LIN {X 0,Y 573.544,Z 345.432,A -85,B 0,C 180,E1 -2260.853,E2 -2260.853} C_VEL
LIN {X 0,Y 573.651,Z 334.309,A -85,B 0,C 180,E1 -2261.446,E2 -2261.446} C_VEL
LIN {X 0,Y 573.758,Z 321.17,A -85,B 0,C 180,E1 -2261.974,E2 -2261.974} C_VEL
LIN {X 0,Y 573.833,Z 308.518,A -85,B 0,C 180,E1 -2262.331,E2 -2262.331} C_VEL
LIN {X 0,Y 573.943,Z 295.311,A -85,B 0,C 180,E1 -2262.553,E2 -2262.553} C_VEL
LIN {X 0,Y 573.985,Z 198.721,A -85,B 0,C 180,E1 -2263.768,E2 -2263.768} C_VEL
LIN {X 0,Y 573.396,Z 194.613,A -85,B 0,C 180,E1 -2263.851,E2 -2263.851} C_VEL
LIN {X 0,Y 573.568,Z 174.153,A -85,B 0,C 180,E1 -2266.722,E2 -2266.722} C_VEL
LIN {X 0,Y 573.786,Z 153.399,A -85,B 0,C 180,E1 -2269.647,E2 -2269.647} C_VEL
LIN {X 0,Y 573.952,Z 134.662,A -85,B 0,C 180,E1 -2272.308,E2 -2272.308} C_VEL
LIN {X 0,Y 573.639,Z 129.359,A -85,B 0,C 180,E1 -2273.082,E2 -2273.082} C_VEL
LIN {X 0,Y 573.228,Z 127.085,A -85,B 0,C 180,E1 -2273.438,E2 -2273.438} C_VEL
LIN {X 0,Y 573.239,Z 127.079,A -85,B 0,C 180,E1 -2276.191,E2 -2276.191} C_VEL
LIN {X 0,Y 573.199,Z 127.081,A -85,B 0,C 180,E1 -2278.567,E2 -2278.567} C_VEL
LIN {X 0,Y 573.219,Z 127.08,A -85,B 0,C 180,E1 -2280.994,E2 -2280.994} C_VEL
LIN {X 0,Y 573.244,Z 127.083,A -85,B 0,C 180,E1 -2283.521,E2 -2283.521} C_VEL
LIN {X 0,Y 573.188,Z 127.082,A -85,B 0,C 180,E1 -2286.054,E2 -2286.054} C_VEL
LIN {X 0,Y 573.23,Z 127.078,A -85,B 0,C 180,E1 -2288.703,E2 -2288.703} C_VEL
LIN {X 0,Y 573.198,Z 127.084,A -85,B 0,C 180,E1 -2291.589,E2 -2291.589} C_VEL
LIN {X 0,Y 573.21,Z 127.081,A -85,B 0,C 180,E1 -2294.673,E2 -2294.673} C_VEL
LIN {X 0,Y 573.203,Z 127.081,A -85,B 0,C 180,E1 -2297.596,E2 -2297.596} C_VEL
LIN {X 0,Y 573.224,Z 127.081,A -85,B 0,C 180,E1 -2300.571,E2 -2300.571} C_VEL
LIN {X 0,Y 573.22,Z 127.083,A -85,B 0,C 180,E1 -2303.075,E2 -2303.075} C_VEL
LIN {X 0,Y 573.221,Z 127.076,A -85,B 0,C 180,E1 -2305.668,E2 -2305.668} C_VEL
LIN {X 0,Y 573.208,Z 127.081,A -85,B 0,C 180,E1 -2308.182,E2 -2308.182} C_VEL
LIN {X 0,Y 573.215,Z 127.087,A -85,B 0,C 180,E1 -2310.631,E2 -2310.631} C_VEL
LIN {X 0,Y 573.195,Z 127.079,A -85,B 0,C 180,E1 -2313.517,E2 -2313.517} C_VEL
LIN {X 0,Y 573.192,Z 127.085,A -85,B 0,C 180,E1 -2316.132,E2 -2316.132} C_VEL
LIN {X 0,Y 573.22,Z 127.077,A -85,B 0,C 180,E1 -2319.172,E2 -2319.172} C_VEL
LIN {X 0,Y 573.2,Z 127.087,A -85,B 0,C 180,E1 -2322.15,E2 -2322.15} C_VEL
LIN {X 0,Y 573.217,Z 127.077,A -85,B 0,C 180,E1 -2325.079,E2 -2325.079} C_VEL
LIN {X 0,Y 573.238,Z 127.082,A -85,B 0,C 180,E1 -2327.97,E2 -2327.97} C_VEL
LIN {X 0,Y 573.221,Z 127.076,A -85,B 0,C 180,E1 -2330.828,E2 -2330.828} C_VEL
LIN {X 0,Y 573.233,Z 127.081,A -85,B 0,C 180,E1 -2333.665,E2 -2333.665} C_VEL
LIN {X 0,Y 573.22,Z 127.085,A -85,B 0,C 180,E1 -2335.781,E2 -2335.781} C_VEL
LIN {X 0,Y 573.312,Z 127.072,A -85,B 0,C 180,E1 -2337.892,E2 -2337.892} C_VEL
LIN {X 0,Y 573.322,Z 127.068,A -85,B 0,C 180,E1 -2340,E2 -2340} C_VEL
LIN {X 0,Y 573.287,Z 127.069,A -85,B 0,C 180,E1 -2342.81,E2 -2342.81} C_VEL
LIN {X 0,Y 573.285,Z 127.075,A -85,B 0,C 180,E1 -2345.628,E2 -2345.628} C_VEL
LIN {X 0,Y 573.25,Z 127.073,A -85,B 0,C 180,E1 -2348.46,E2 -2348.46} C_VEL
LIN {X 0,Y 573.275,Z 127.079,A -85,B 0,C 180,E1 -2351.311,E2 -2351.311} C_VEL
LIN {X 0,Y 573.265,Z 127.071,A -85,B 0,C 180,E1 -2354.416,E2 -2354.416} C_VEL
LIN {X 0,Y 573.249,Z 127.083,A -85,B 0,C 180,E1 -2357.111,E2 -2357.111} C_VEL
LIN {X 0,Y 573.238,Z 127.075,A -85,B 0,C 180,E1 -2360.077,E2 -2360.077} C_VEL
LIN {X 0,Y 573.223,Z 127.077,A -85,B 0,C 180,E1 -2362.338,E2 -2362.338} C_VEL
LIN {X 0,Y 573.215,Z 127.08,A -85,B 0,C 180,E1 -2364.351,E2 -2364.351} C_VEL
LIN {X 0,Y 572.581,Z 127.165,A -85,B 0,C 180,E1 -2364.937,E2 -2364.937} C_VEL
LIN {X 0,Y 569.758,Z 127.517,A -85,B 0,C 180,E1 -2365.889,E2 -2365.889} C_VEL
LIN {X 0,Y 567.346,Z 127.817,A -85,B 0,C 180,E1 -2366.655,E2 -2366.655} C_VEL
LIN {X 0,Y 566.293,Z 127.943,A -85,B 0,C 180,E1 -2367.246,E2 -2367.246} C_VEL
LIN {X 0,Y 566.2,Z 127.952,A -85,B 0,C 180,E1 -2367.446,E2 -2367.446} C_VEL
LIN {X 0,Y 566.198,Z 127.952,A -85,B 0,C 180,E1 -2369.769,E2 -2369.769} C_VEL
LIN {X 0,Y 566.203,Z 127.958,A -85,B 0,C 180,E1 -2372.429,E2 -2372.429} C_VEL
LIN {X 0,Y 566.18,Z 127.957,A -85,B 0,C 180,E1 -2374.989,E2 -2374.989} C_VEL
LIN {X 0,Y 566.196,Z 127.953,A -85,B 0,C 180,E1 -2377.46,E2 -2377.46} C_VEL
LIN {X 0,Y 566.206,Z 127.959,A -85,B 0,C 180,E1 -2380.199,E2 -2380.199} C_VEL
LIN {X 0,Y 566.201,Z 127.954,A -85,B 0,C 180,E1 -2383.054,E2 -2383.054} C_VEL
LIN {X 0,Y 566.197,Z 127.961,A -85,B 0,C 180,E1 -2386.048,E2 -2386.048} C_VEL
LIN {X 0,Y 566.205,Z 127.954,A -85,B 0,C 180,E1 -2388.863,E2 -2388.863} C_VEL
LIN {X 0,Y 566.255,Z 128.085,A -85,B 0,C 180,E1 -2390.913,E2 -2390.913} C_VEL
LIN {X 0,Y 566.427,Z 135.904,A -85,B 0,C 180,E1 -2392.333,E2 -2392.333} C_VEL
LIN {X 0,Y 566.298,Z 148.953,A -85,B 0,C 180,E1 -2394.69,E2 -2394.69} C_VEL
LIN {X 0,Y 566.209,Z 156.367,A -85,B 0,C 180,E1 -2396.044,E2 -2396.044} C_VEL
LIN {X 0,Y 567.178,Z 162.749,A -85,B 0,C 180,E1 -2396.16,E2 -2396.16} C_VEL
LIN {X 0,Y 566.94,Z 263.602,A -85,B 0,C 180,E1 -2397.461,E2 -2397.461} C_VEL
LIN {X 0,Y 566.855,Z 276.85,A -85,B 0,C 180,E1 -2397.783,E2 -2397.783} C_VEL
LIN {X 0,Y 566.716,Z 289.665,A -85,B 0,C 180,E1 -2398.245,E2 -2398.245} C_VEL
LIN {X 0,Y 566.54,Z 302.13,A -85,B 0,C 180,E1 -2398.864,E2 -2398.864} C_VEL
LIN {X 0,Y 566.388,Z 314.001,A -85,B 0,C 180,E1 -2399.626,E2 -2399.626} C_VEL
LIN {X 0,Y 566.304,Z 324.474,A -85,B 0,C 180,E1 -2400.477,E2 -2400.477} C_VEL
LIN {X 0,Y 566.162,Z 334.165,A -85,B 0,C 180,E1 -2401.451,E2 -2401.451} C_VEL
LIN {X 0,Y 566.061,Z 342.273,A -85,B 0,C 180,E1 -2402.453,E2 -2402.453} C_VEL
LIN {X 0,Y 565.981,Z 349.966,A -85,B 0,C 180,E1 -2403.646,E2 -2403.646} C_VEL
LIN {X 0,Y 565.937,Z 355.053,A -85,B 0,C 180,E1 -2404.632,E2 -2404.632} C_VEL
LIN {X 0,Y 565.893,Z 359.794,A -85,B 0,C 180,E1 -2405.805,E2 -2405.805} C_VEL
LIN {X 0,Y 565.882,Z 362.787,A -85,B 0,C 180,E1 -2406.786,E2 -2406.786} C_VEL
LIN {X 0,Y 565.831,Z 365.533,A -85,B 0,C 180,E1 -2408.123,E2 -2408.123} C_VEL
LIN {X 0,Y 565.873,Z 366.478,A -85,B 0,C 180,E1 -2408.889,E2 -2408.889} C_VEL
LIN {X 0,Y 565.833,Z 366.918,A -85,B 0,C 180,E1 -2409.649,E2 -2409.649} C_VEL
LIN {X 0,Y 565.868,Z 366.812,A -85,B 0,C 180,E1 -2410.717,E2 -2410.717} C_VEL
LIN {X 0,Y 565.835,Z 365.622,A -85,B 0,C 180,E1 -2411.91,E2 -2411.91} C_VEL
LIN {X 0,Y 565.853,Z 363.526,A -85,B 0,C 180,E1 -2413.008,E2 -2413.008} C_VEL
LIN {X 0,Y 565.892,Z 360.284,A -85,B 0,C 180,E1 -2414.144,E2 -2414.144} C_VEL
LIN {X 0,Y 565.959,Z 355.817,A -85,B 0,C 180,E1 -2415.289,E2 -2415.289} C_VEL
LIN {X 0,Y 566.005,Z 349.441,A -85,B 0,C 180,E1 -2416.537,E2 -2416.537} C_VEL
LIN {X 0,Y 566.049,Z 342.308,A -85,B 0,C 180,E1 -2417.633,E2 -2417.633} C_VEL
LIN {X 0,Y 566.158,Z 333.501,A -85,B 0,C 180,E1 -2418.712,E2 -2418.712} C_VEL
LIN {X 0,Y 566.305,Z 324.259,A -85,B 0,C 180,E1 -2419.633,E2 -2419.633} C_VEL
LIN {X 0,Y 566.409,Z 314.235,A -85,B 0,C 180,E1 -2420.447,E2 -2420.447} C_VEL
LIN {X 0,Y 566.58,Z 303.086,A -85,B 0,C 180,E1 -2421.17,E2 -2421.17} C_VEL
LIN {X 0,Y 566.709,Z 290.648,A -85,B 0,C 180,E1 -2421.801,E2 -2421.801} C_VEL
LIN {X 0,Y 566.807,Z 278.481,A -85,B 0,C 180,E1 -2422.26,E2 -2422.26} C_VEL
LIN {X 0,Y 566.933,Z 265.223,A -85,B 0,C 180,E1 -2422.597,E2 -2422.597} C_VEL
LIN {X 0,Y 567,Z 245.47,A -85,B 0,C 180,E1 -2422.88,E2 -2422.88} C_VEL
LIN {X 0,Y 567.1,Z 161.979,A -85,B 0,C 180,E1 -2423.942,E2 -2423.942} C_VEL
LIN {X 0,Y 566.216,Z 156.317,A -85,B 0,C 180,E1 -2424.056,E2 -2424.056} C_VEL
LIN {X 0,Y 566.36,Z 141.28,A -85,B 0,C 180,E1 -2426.799,E2 -2426.799} C_VEL
LIN {X 0,Y 566.396,Z 129.601,A -85,B 0,C 180,E1 -2428.934,E2 -2428.934} C_VEL
LIN {X 0,Y 566.137,Z 127.965,A -85,B 0,C 180,E1 -2429.289,E2 -2429.289} C_VEL
LIN {X 0,Y 566.138,Z 127.962,A -85,B 0,C 180,E1 -2430.711,E2 -2430.711} C_VEL
LIN {X 0,Y 566.233,Z 127.949,A -85,B 0,C 180,E1 -2432.846,E2 -2432.846} C_VEL
LIN {X 0,Y 566.231,Z 127.953,A -85,B 0,C 180,E1 -2435.699,E2 -2435.699} C_VEL
LIN {X 0,Y 566.18,Z 127.955,A -85,B 0,C 180,E1 -2438.567,E2 -2438.567} C_VEL
LIN {X 0,Y 566.187,Z 127.957,A -85,B 0,C 180,E1 -2441.456,E2 -2441.456} C_VEL
LIN {X 0,Y 566.198,Z 127.952,A -85,B 0,C 180,E1 -2444.494,E2 -2444.494} C_VEL
LIN {X 0,Y 566.151,Z 127.962,A -85,B 0,C 180,E1 -2447.333,E2 -2447.333} C_VEL
LIN {X 0,Y 566.138,Z 127.959,A -85,B 0,C 180,E1 -2450.34,E2 -2450.34} C_VEL
LIN {X 0,Y 566.131,Z 127.96,A -85,B 0,C 180,E1 -2452.634,E2 -2452.634} C_VEL
LIN {X 0,Y 566.141,Z 127.962,A -85,B 0,C 180,E1 -2455.014,E2 -2455.014} C_VEL
LIN {X 0,Y 566.152,Z 127.966,A -85,B 0,C 180,E1 -2457.343,E2 -2457.343} C_VEL
LIN {X 0,Y 566.141,Z 127.962,A -85,B 0,C 180,E1 -2459.773,E2 -2459.773} C_VEL
LIN {X 0,Y 566.167,Z 127.955,A -85,B 0,C 180,E1 -2462.425,E2 -2462.425} C_VEL
LIN {X 0,Y 566.15,Z 127.964,A -85,B 0,C 180,E1 -2464.986,E2 -2464.986} C_VEL
LIN {X 0,Y 566.175,Z 127.959,A -85,B 0,C 180,E1 -2467.463,E2 -2467.463} C_VEL
LIN {X 0,Y 566.162,Z 127.956,A -85,B 0,C 180,E1 -2470.203,E2 -2470.203} C_VEL
LIN {X 0,Y 566.144,Z 127.967,A -85,B 0,C 180,E1 -2473.06,E2 -2473.06} C_VEL
LIN {X 0,Y 566.153,Z 127.957,A -85,B 0,C 180,E1 -2476.054,E2 -2476.054} C_VEL
LIN {X 0,Y 566.14,Z 127.969,A -85,B 0,C 180,E1 -2478.858,E2 -2478.858} C_VEL
LIN {X 0,Y 566.169,Z 127.955,A -85,B 0,C 180,E1 -2481.636,E2 -2481.636} C_VEL
LIN {X 0,Y 566.132,Z 127.963,A -85,B 0,C 180,E1 -2484.306,E2 -2484.306} C_VEL
LIN {X 0,Y 566.162,Z 127.962,A -85,B 0,C 180,E1 -2486.895,E2 -2486.895} C_VEL
LIN {X 0,Y 566.149,Z 127.958,A -85,B 0,C 180,E1 -2489.406,E2 -2489.406} C_VEL
LIN {X 0,Y 566.141,Z 127.959,A -85,B 0,C 180,E1 -2491.854,E2 -2491.854} C_VEL
LIN {X 0,Y 566.177,Z 127.96,A -85,B 0,C 180,E1 -2494.25,E2 -2494.25} C_VEL
LIN {X 0,Y 566.149,Z 127.962,A -85,B 0,C 180,E1 -2496.726,E2 -2496.726} C_VEL
LIN {X 0,Y 566.183,Z 127.955,A -85,B 0,C 180,E1 -2498.902,E2 -2498.902} C_VEL
LIN {X 0,Y 566.153,Z 127.961,A -85,B 0,C 180,E1 -2501.921,E2 -2501.921} C_VEL
LIN {X 0,Y 566.152,Z 127.958,A -85,B 0,C 180,E1 -2504.89,E2 -2504.89} C_VEL
LIN {X 0,Y 566.149,Z 127.958,A -85,B 0,C 180,E1 -2507.089,E2 -2507.089} C_VEL
LIN {X 0,Y 566.213,Z 127.95,A -85,B 0,C 180,E1 -2509.27,E2 -2509.27} C_VEL
LIN {X 0,Y 566.19,Z 127.96,A -85,B 0,C 180,E1 -2512.153,E2 -2512.153} C_VEL
LIN {X 0,Y 566.251,Z 127.945,A -85,B 0,C 180,E1 -2515.016,E2 -2515.016} C_VEL
LIN {X 0,Y 566.281,Z 127.951,A -85,B 0,C 180,E1 -2517.867,E2 -2517.867} C_VEL
LIN {X 0,Y 566.289,Z 127.947,A -85,B 0,C 180,E1 -2520,E2 -2520} C_VEL
LIN {X 0,Y 566.24,Z 127.946,A -85,B 0,C 180,E1 -2522.846,E2 -2522.846} C_VEL
LIN {X 0,Y 566.24,Z 127.956,A -85,B 0,C 180,E1 -2525.699,E2 -2525.699} C_VEL
LIN {X 0,Y 566.19,Z 127.952,A -85,B 0,C 180,E1 -2528.567,E2 -2528.567} C_VEL
LIN {X 0,Y 566.244,Z 127.954,A -85,B 0,C 180,E1 -2531.455,E2 -2531.455} C_VEL
LIN {X 0,Y 566.182,Z 127.953,A -85,B 0,C 180,E1 -2534.483,E2 -2534.483} C_VEL
LIN {X 0,Y 566.164,Z 127.964,A -85,B 0,C 180,E1 -2537.333,E2 -2537.333} C_VEL
LIN {X 0,Y 566.197,Z 127.957,A -85,B 0,C 180,E1 -2539.581,E2 -2539.581} C_VEL
LIN {X 0,Y 566.154,Z 127.959,A -85,B 0,C 180,E1 -2541.865,E2 -2541.865} C_VEL
LIN {X 0,Y 566.184,Z 127.96,A -85,B 0,C 180,E1 -2545.021,E2 -2545.021} C_VEL
LIN {X 0,Y 566.166,Z 127.962,A -85,B 0,C 180,E1 -2547.342,E2 -2547.342} C_VEL
LIN {X 0,Y 566.155,Z 127.958,A -85,B 0,C 180,E1 -2549.772,E2 -2549.772} C_VEL
LIN {X 0,Y 566.197,Z 127.953,A -85,B 0,C 180,E1 -2552.428,E2 -2552.428} C_VEL
LIN {X 0,Y 566.171,Z 127.964,A -85,B 0,C 180,E1 -2554.987,E2 -2554.987} C_VEL
LIN {X 0,Y 566.195,Z 127.954,A -85,B 0,C 180,E1 -2557.461,E2 -2557.461} C_VEL
LIN {X 0,Y 566.21,Z 127.951,A -85,B 0,C 180,E1 -2560.199,E2 -2560.199} C_VEL
LIN {X 0,Y 566.182,Z 127.958,A -85,B 0,C 180,E1 -2563.056,E2 -2563.056} C_VEL
LIN {X 0,Y 566.16,Z 127.957,A -85,B 0,C 180,E1 -2566.053,E2 -2566.053} C_VEL
LIN {X 0,Y 566.206,Z 127.952,A -85,B 0,C 180,E1 -2569.215,E2 -2569.215} C_VEL
LIN {X 0,Y 566.177,Z 127.954,A -85,B 0,C 180,E1 -2571.636,E2 -2571.636} C_VEL
LIN {X 0,Y 566.145,Z 127.965,A -85,B 0,C 180,E1 -2574.306,E2 -2574.306} C_VEL
LIN {X 0,Y 566.199,Z 127.954,A -85,B 0,C 180,E1 -2576.896,E2 -2576.896} C_VEL
LIN {X 0,Y 566.171,Z 127.956,A -85,B 0,C 180,E1 -2579.406,E2 -2579.406} C_VEL
LIN {X 0,Y 566.155,Z 127.961,A -85,B 0,C 180,E1 -2581.854,E2 -2581.854} C_VEL
LIN {X 0,Y 566.194,Z 127.962,A -85,B 0,C 180,E1 -2584.25,E2 -2584.25} C_VEL
LIN {X 0,Y 566.188,Z 128.083,A -85,B 0,C 180,E1 -2586.426,E2 -2586.426} C_VEL
LIN {X 0,Y 567,Z 133.221,A -85,B 0,C 180,E1 -2587.21,E2 -2587.21} C_VEL
LIN {X 0,Y 566.834,Z 152.953,A -85,B 0,C 180,E1 -2590.064,E2 -2590.064} C_VEL
LIN {X 0,Y 566.589,Z 174.356,A -85,B 0,C 180,E1 -2593.111,E2 -2593.111} C_VEL
LIN {X 0,Y 566.391,Z 194.611,A -85,B 0,C 180,E1 -2595.974,E2 -2595.974} C_VEL
LIN {X 0,Y 567.156,Z 200.489,A -85,B 0,C 180,E1 -2596.085,E2 -2596.085} C_VEL
LIN {X 0,Y 566.969,Z 302.934,A -85,B 0,C 180,E1 -2597.403,E2 -2597.403} C_VEL
LIN {X 0,Y 566.84,Z 316.21,A -85,B 0,C 180,E1 -2597.718,E2 -2597.718} C_VEL
LIN {X 0,Y 566.743,Z 328.372,A -85,B 0,C 180,E1 -2598.148,E2 -2598.148} C_VEL
LIN {X 0,Y 566.604,Z 340.235,A -85,B 0,C 180,E1 -2598.712,E2 -2598.712} C_VEL
LIN {X 0,Y 566.439,Z 352.193,A -85,B 0,C 180,E1 -2599.455,E2 -2599.455} C_VEL
LIN {X 0,Y 566.325,Z 362.602,A -85,B 0,C 180,E1 -2600.265,E2 -2600.265} C_VEL
LIN {X 0,Y 566.207,Z 371.111,A -85,B 0,C 180,E1 -2601.074,E2 -2601.074} C_VEL
LIN {X 0,Y 566.113,Z 378.959,A -85,B 0,C 180,E1 -2601.971,E2 -2601.971} C_VEL
LIN {X 0,Y 566.004,Z 386.621,A -85,B 0,C 180,E1 -2603.046,E2 -2603.046} C_VEL
LIN {X 0,Y 566.004,Z 393.679,A -85,B 0,C 180,E1 -2604.299,E2 -2604.299} C_VEL
LIN {X 0,Y 565.933,Z 398.372,A -85,B 0,C 180,E1 -2605.37,E2 -2605.37} C_VEL
LIN {X 0,Y 565.927,Z 401.958,A -85,B 0,C 180,E1 -2606.44,E2 -2606.44} C_VEL
LIN {X 0,Y 565.878,Z 403.807,A -85,B 0,C 180,E1 -2607.152,E2 -2607.152} C_VEL
LIN {X 0,Y 565.846,Z 406.184,A -85,B 0,C 180,E1 -2608.576,E2 -2608.576} C_VEL
LIN {X 0,Y 565.839,Z 407,A -85,B 0,C 180,E1 -2610,E2 -2610} C_VEL
LIN {X 0,Y 565.846,Z 406.185,A -85,B 0,C 180,E1 -2611.423,E2 -2611.423} C_VEL
LIN {X 0,Y 565.878,Z 403.81,A -85,B 0,C 180,E1 -2612.847,E2 -2612.847} C_VEL
LIN {X 0,Y 565.926,Z 400.896,A -85,B 0,C 180,E1 -2613.916,E2 -2613.916} C_VEL
LIN {X 0,Y 565.878,Z 396.949,A -85,B 0,C 180,E1 -2614.987,E2 -2614.987} C_VEL
LIN {X 0,Y 566.002,Z 391.868,A -85,B 0,C 180,E1 -2616.058,E2 -2616.058} C_VEL
LIN {X 0,Y 566.04,Z 385.468,A -85,B 0,C 180,E1 -2617.132,E2 -2617.132} C_VEL
LIN {X 0,Y 566.134,Z 377.478,A -85,B 0,C 180,E1 -2618.208,E2 -2618.208} C_VEL
LIN {X 0,Y 566.229,Z 369.334,A -85,B 0,C 180,E1 -2619.105,E2 -2619.105} C_VEL
LIN {X 0,Y 566.347,Z 359.399,A -85,B 0,C 180,E1 -2620.005,E2 -2620.005} C_VEL
LIN {X 0,Y 566.536,Z 348.291,A -85,B 0,C 180,E1 -2620.807,E2 -2620.807} C_VEL
LIN {X 0,Y 566.613,Z 337.173,A -85,B 0,C 180,E1 -2621.447,E2 -2621.447} C_VEL
LIN {X 0,Y 566.745,Z 324.979,A -85,B 0,C 180,E1 -2621.988,E2 -2621.988} C_VEL
LIN {X 0,Y 566.914,Z 312.175,A -85,B 0,C 180,E1 -2622.393,E2 -2622.393} C_VEL
LIN {X 0,Y 567.007,Z 300.106,A -85,B 0,C 180,E1 -2622.641,E2 -2622.641} C_VEL
LIN {X 0,Y 567.053,Z 199.28,A -85,B 0,C 180,E1 -2623.933,E2 -2623.933} C_VEL
LIN {X 0,Y 566.391,Z 194.613,A -85,B 0,C 180,E1 -2624.025,E2 -2624.025} C_VEL
LIN {X 0,Y 566.588,Z 174.331,A -85,B 0,C 180,E1 -2626.888,E2 -2626.888} C_VEL
LIN {X 0,Y 566.855,Z 151.538,A -85,B 0,C 180,E1 -2630.124,E2 -2630.124} C_VEL
LIN {X 0,Y 566.986,Z 133.053,A -85,B 0,C 180,E1 -2632.79,E2 -2632.79} C_VEL
LIN {X 0,Y 566.195,Z 127.961,A -85,B 0,C 180,E1 -2633.598,E2 -2633.598} C_VEL
LIN {X 0,Y 566.186,Z 127.955,A -85,B 0,C 180,E1 -2636.543,E2 -2636.543} C_VEL
LIN {X 0,Y 566.171,Z 127.964,A -85,B 0,C 180,E1 -2639.771,E2 -2639.771} C_VEL
LIN {X 0,Y 566.193,Z 127.953,A -85,B 0,C 180,E1 -2642.428,E2 -2642.428} C_VEL
LIN {X 0,Y 566.166,Z 127.958,A -85,B 0,C 180,E1 -2644.987,E2 -2644.987} C_VEL
LIN {X 0,Y 566.191,Z 127.961,A -85,B 0,C 180,E1 -2647.462,E2 -2647.462} C_VEL
LIN {X 0,Y 566.196,Z 127.952,A -85,B 0,C 180,E1 -2650.2,E2 -2650.2} C_VEL
LIN {X 0,Y 566.178,Z 127.962,A -85,B 0,C 180,E1 -2653.057,E2 -2653.057} C_VEL
LIN {X 0,Y 566.156,Z 127.957,A -85,B 0,C 180,E1 -2656.053,E2 -2656.053} C_VEL
LIN {X 0,Y 566.143,Z 127.966,A -85,B 0,C 180,E1 -2658.857,E2 -2658.857} C_VEL
LIN {X 0,Y 566.159,Z 127.958,A -85,B 0,C 180,E1 -2661.449,E2 -2661.449} C_VEL
LIN {X 0,Y 566.154,Z 127.957,A -85,B 0,C 180,E1 -2663.793,E2 -2663.793} C_VEL
LIN {X 0,Y 566.16,Z 127.958,A -85,B 0,C 180,E1 -2666.274,E2 -2666.274} C_VEL
LIN {X 0,Y 566.171,Z 127.96,A -85,B 0,C 180,E1 -2668.928,E2 -2668.928} C_VEL
LIN {X 0,Y 566.141,Z 127.959,A -85,B 0,C 180,E1 -2671.853,E2 -2671.853} C_VEL
LIN {X 0,Y 566.174,Z 127.959,A -85,B 0,C 180,E1 -2674.249,E2 -2674.249} C_VEL
LIN {X 0,Y 566.15,Z 127.961,A -85,B 0,C 180,E1 -2676.725,E2 -2676.725} C_VEL
LIN {X 0,Y 566.184,Z 127.955,A -85,B 0,C 180,E1 -2678.901,E2 -2678.901} C_VEL
LIN {X 0,Y 566.156,Z 127.961,A -85,B 0,C 180,E1 -2681.92,E2 -2681.92} C_VEL
LIN {X 0,Y 566.182,Z 127.954,A -85,B 0,C 180,E1 -2684.89,E2 -2684.89} C_VEL
LIN {X 0,Y 566.182,Z 127.958,A -85,B 0,C 180,E1 -2687.817,E2 -2687.817} C_VEL
LIN {X 0,Y 566.166,Z 127.965,A -85,B 0,C 180,E1 -2689.992,E2 -2689.992} C_VEL
LIN {X 0,Y 566.193,Z 127.957,A -85,B 0,C 180,E1 -2692.152,E2 -2692.152} C_VEL
LIN {X 0,Y 566.259,Z 127.944,A -85,B 0,C 180,E1 -2695.016,E2 -2695.016} C_VEL
LIN {X 0,Y 566.283,Z 127.948,A -85,B 0,C 180,E1 -2697.866,E2 -2697.866} C_VEL
LIN {X 0,Y 566.29,Z 127.943,A -85,B 0,C 180,E1 -2700,E2 -2700} C_VEL
LIN {X 0,Y 566.256,Z 127.945,A -85,B 0,C 180,E1 -2702.845,E2 -2702.845} C_VEL
LIN {X 0,Y 566.252,Z 127.95,A -85,B 0,C 180,E1 -2705.698,E2 -2705.698} C_VEL
LIN {X 0,Y 566.202,Z 127.952,A -85,B 0,C 180,E1 -2708.566,E2 -2708.566} C_VEL
LIN {X 0,Y 566.245,Z 127.953,A -85,B 0,C 180,E1 -2711.454,E2 -2711.454} C_VEL
LIN {X 0,Y 566.221,Z 127.949,A -85,B 0,C 180,E1 -2714.499,E2 -2714.499} C_VEL
LIN {X 0,Y 566.19,Z 127.958,A -85,B 0,C 180,E1 -2717.331,E2 -2717.331} C_VEL
LIN {X 0,Y 566.202,Z 127.953,A -85,B 0,C 180,E1 -2719.58,E2 -2719.58} C_VEL
LIN {X 0,Y 566.188,Z 127.952,A -85,B 0,C 180,E1 -2721.862,E2 -2721.862} C_VEL
LIN {X 0,Y 566.185,Z 127.96,A -85,B 0,C 180,E1 -2725.022,E2 -2725.022} C_VEL
LIN {X 0,Y 566.2,Z 127.952,A -85,B 0,C 180,E1 -2727.446,E2 -2727.446} C_VEL
LIN {X 0,Y 565.511,Z 128.039,A -85,B 0,C 180,E1 -2728.04,E2 -2728.04} C_VEL
LIN {X 0,Y 562.647,Z 128.4,A -85,B 0,C 180,E1 -2729.004,E2 -2729.004} C_VEL
LIN {X 0,Y 560.243,Z 128.697,A -85,B 0,C 180,E1 -2729.779,E2 -2729.779} C_VEL
LIN {X 0,Y 559.217,Z 128.827,A -85,B 0,C 180,E1 -2730.378,E2 -2730.378} C_VEL
LIN {X 0,Y 559.136,Z 128.833,A -85,B 0,C 180,E1 -2730.581,E2 -2730.581} C_VEL
LIN {X 0,Y 559.152,Z 128.837,A -85,B 0,C 180,E1 -2732.715,E2 -2732.715} C_VEL
LIN {X 0,Y 559.127,Z 128.834,A -85,B 0,C 180,E1 -2735.324,E2 -2735.324} C_VEL
LIN {X 0,Y 559.133,Z 128.837,A -85,B 0,C 180,E1 -2738.017,E2 -2738.017} C_VEL
LIN {X 0,Y 559.157,Z 128.833,A -85,B 0,C 180,E1 -2740.812,E2 -2740.812} C_VEL
LIN {X 0,Y 559.146,Z 128.832,A -85,B 0,C 180,E1 -2743.196,E2 -2743.196} C_VEL
LIN {X 0,Y 559.158,Z 128.838,A -85,B 0,C 180,E1 -2746.268,E2 -2746.268} C_VEL
LIN {X 0,Y 559.173,Z 128.83,A -85,B 0,C 180,E1 -2749.189,E2 -2749.189} C_VEL
LIN {X 0,Y 559.213,Z 128.974,A -85,B 0,C 180,E1 -2750.837,E2 -2750.837} C_VEL
LIN {X 0,Y 559.462,Z 134.221,A -85,B 0,C 180,E1 -2751.797,E2 -2751.797} C_VEL
LIN {X 0,Y 559.358,Z 147.778,A -85,B 0,C 180,E1 -2754.25,E2 -2754.25} C_VEL
LIN {X 0,Y 559.177,Z 156.557,A -85,B 0,C 180,E1 -2755.873,E2 -2755.873} C_VEL
LIN {X 0,Y 560.318,Z 163.963,A -85,B 0,C 180,E1 -2755.999,E2 -2755.999} C_VEL
LIN {X 0,Y 560.011,Z 263.471,A -85,B 0,C 180,E1 -2757.298,E2 -2757.298} C_VEL
LIN {X 0,Y 559.927,Z 276.907,A -85,B 0,C 180,E1 -2757.628,E2 -2757.628} C_VEL
LIN {X 0,Y 559.766,Z 289.066,A -85,B 0,C 180,E1 -2758.069,E2 -2758.069} C_VEL
LIN {X 0,Y 559.566,Z 300.986,A -85,B 0,C 180,E1 -2758.655,E2 -2758.655} C_VEL
LIN {X 0,Y 559.419,Z 312.894,A -85,B 0,C 180,E1 -2759.416,E2 -2759.416} C_VEL
LIN {X 0,Y 559.289,Z 322.601,A -85,B 0,C 180,E1 -2760.187,E2 -2760.187} C_VEL
LIN {X 0,Y 559.168,Z 331.632,A -85,B 0,C 180,E1 -2761.06,E2 -2761.06} C_VEL
LIN {X 0,Y 559.033,Z 340.227,A -85,B 0,C 180,E1 -2762.082,E2 -2762.082} C_VEL
LIN {X 0,Y 558.928,Z 347.962,A -85,B 0,C 180,E1 -2763.221,E2 -2763.221} C_VEL
LIN {X 0,Y 558.861,Z 353.76,A -85,B 0,C 180,E1 -2764.287,E2 -2764.287} C_VEL
LIN {X 0,Y 558.837,Z 358.853,A -85,B 0,C 180,E1 -2765.48,E2 -2765.48} C_VEL
LIN {X 0,Y 558.799,Z 362.556,A -85,B 0,C 180,E1 -2766.651,E2 -2766.651} C_VEL
LIN {X 0,Y 558.745,Z 365.116,A -85,B 0,C 180,E1 -2767.831,E2 -2767.831} C_VEL
LIN {X 0,Y 558.755,Z 366.188,A -85,B 0,C 180,E1 -2768.607,E2 -2768.607} C_VEL
LIN {X 0,Y 558.742,Z 366.822,A -85,B 0,C 180,E1 -2769.379,E2 -2769.379} C_VEL
LIN {X 0,Y 558.765,Z 366.875,A -85,B 0,C 180,E1 -2770.617,E2 -2770.617} C_VEL
LIN {X 0,Y 558.73,Z 365.977,A -85,B 0,C 180,E1 -2771.672,E2 -2771.672} C_VEL
LIN {X 0,Y 558.762,Z 363.823,A -85,B 0,C 180,E1 -2772.922,E2 -2772.922} C_VEL
LIN {X 0,Y 558.796,Z 361.114,A -85,B 0,C 180,E1 -2773.937,E2 -2773.937} C_VEL
LIN {X 0,Y 558.885,Z 357.083,A -85,B 0,C 180,E1 -2775.061,E2 -2775.061} C_VEL
LIN {X 0,Y 558.918,Z 350.868,A -85,B 0,C 180,E1 -2776.363,E2 -2776.363} C_VEL
LIN {X 0,Y 558.98,Z 344.068,A -85,B 0,C 180,E1 -2777.474,E2 -2777.474} C_VEL
LIN {X 0,Y 559.093,Z 335.53,A -85,B 0,C 180,E1 -2778.595,E2 -2778.595} C_VEL
LIN {X 0,Y 559.192,Z 326.998,A -85,B 0,C 180,E1 -2779.5,E2 -2779.5} C_VEL
LIN {X 0,Y 559.375,Z 316.34,A -85,B 0,C 180,E1 -2780.417,E2 -2780.417} C_VEL
LIN {X 0,Y 559.572,Z 305.784,A -85,B 0,C 180,E1 -2781.15,E2 -2781.15} C_VEL
LIN {X 0,Y 559.725,Z 294.169,A -85,B 0,C 180,E1 -2781.789,E2 -2781.789} C_VEL
LIN {X 0,Y 559.825,Z 281.511,A -85,B 0,C 180,E1 -2782.312,E2 -2782.312} C_VEL
LIN {X 0,Y 559.96,Z 268.649,A -85,B 0,C 180,E1 -2782.686,E2 -2782.686} C_VEL
LIN {X 0,Y 560.002,Z 255.436,A -85,B 0,C 180,E1 -2782.916,E2 -2782.916} C_VEL
LIN {X 0,Y 560.262,Z 162.924,A -85,B 0,C 180,E1 -2784.105,E2 -2784.105} C_VEL
LIN {X 0,Y 559.22,Z 156.541,A -85,B 0,C 180,E1 -2784.23,E2 -2784.23} C_VEL
LIN {X 0,Y 559.364,Z 140.788,A -85,B 0,C 180,E1 -2787.119,E2 -2787.119} C_VEL
LIN {X 0,Y 559.425,Z 131,A -85,B 0,C 180,E1 -2788.92,E2 -2788.92} C_VEL
LIN {X 0,Y 559.108,Z 128.842,A -85,B 0,C 180,E1 -2789.37,E2 -2789.37} C_VEL
LIN {X 0,Y 559.095,Z 128.84,A -85,B 0,C 180,E1 -2790.72,E2 -2790.72} C_VEL
LIN {X 0,Y 559.201,Z 128.825,A -85,B 0,C 180,E1 -2792.882,E2 -2792.882} C_VEL
LIN {X 0,Y 559.2,Z 128.83,A -85,B 0,C 180,E1 -2795.771,E2 -2795.771} C_VEL
LIN {X 0,Y 559.145,Z 128.83,A -85,B 0,C 180,E1 -2798.675,E2 -2798.675} C_VEL
LIN {X 0,Y 559.149,Z 128.836,A -85,B 0,C 180,E1 -2801.602,E2 -2801.602} C_VEL
LIN {X 0,Y 559.148,Z 128.83,A -85,B 0,C 180,E1 -2804.576,E2 -2804.576} C_VEL
LIN {X 0,Y 559.104,Z 128.844,A -85,B 0,C 180,E1 -2807.559,E2 -2807.559} C_VEL
LIN {X 0,Y 559.101,Z 128.835,A -85,B 0,C 180,E1 -2810.608,E2 -2810.608} C_VEL
LIN {X 0,Y 559.091,Z 128.845,A -85,B 0,C 180,E1 -2813.418,E2 -2813.418} C_VEL
LIN {X 0,Y 559.136,Z 128.832,A -85,B 0,C 180,E1 -2816.1,E2 -2816.1} C_VEL
LIN {X 0,Y 559.094,Z 128.837,A -85,B 0,C 180,E1 -2818.534,E2 -2818.534} C_VEL
LIN {X 0,Y 559.112,Z 128.843,A -85,B 0,C 180,E1 -2821.268,E2 -2821.268} C_VEL
LIN {X 0,Y 559.135,Z 128.832,A -85,B 0,C 180,E1 -2823.945,E2 -2823.945} C_VEL
LIN {X 0,Y 559.107,Z 128.844,A -85,B 0,C 180,E1 -2827.112,E2 -2827.112} C_VEL
LIN {X 0,Y 559.122,Z 128.833,A -85,B 0,C 180,E1 -2829.938,E2 -2829.938} C_VEL
LIN {X 0,Y 559.109,Z 128.84,A -85,B 0,C 180,E1 -2832.749,E2 -2832.749} C_VEL
LIN {X 0,Y 559.121,Z 128.833,A -85,B 0,C 180,E1 -2835.765,E2 -2835.765} C_VEL
LIN {X 0,Y 559.095,Z 128.837,A -85,B 0,C 180,E1 -2838.224,E2 -2838.224} C_VEL
LIN {X 0,Y 559.165,Z 128.831,A -85,B 0,C 180,E1 -2841.194,E2 -2841.194} C_VEL
LIN {X 0,Y 559.111,Z 128.834,A -85,B 0,C 180,E1 -2843.788,E2 -2843.788} C_VEL
LIN {X 0,Y 559.123,Z 128.838,A -85,B 0,C 180,E1 -2846.423,E2 -2846.423} C_VEL
LIN {X 0,Y 559.135,Z 128.835,A -85,B 0,C 180,E1 -2848.98,E2 -2848.98} C_VEL
LIN {X 0,Y 559.103,Z 128.835,A -85,B 0,C 180,E1 -2851.632,E2 -2851.632} C_VEL
LIN {X 0,Y 559.147,Z 128.831,A -85,B 0,C 180,E1 -2853.902,E2 -2853.902} C_VEL
LIN {X 0,Y 559.092,Z 128.838,A -85,B 0,C 180,E1 -2857.066,E2 -2857.066} C_VEL
LIN {X 0,Y 559.108,Z 128.835,A -85,B 0,C 180,E1 -2859.393,E2 -2859.393} C_VEL
LIN {X 0,Y 559.112,Z 128.841,A -85,B 0,C 180,E1 -2862.442,E2 -2862.442} C_VEL
LIN {X 0,Y 559.155,Z 128.829,A -85,B 0,C 180,E1 -2865.441,E2 -2865.441} C_VEL
LIN {X 0,Y 559.15,Z 128.832,A -85,B 0,C 180,E1 -2868.637,E2 -2868.637} C_VEL
LIN {X 0,Y 559.154,Z 128.83,A -85,B 0,C 180,E1 -2871.326,E2 -2871.326} C_VEL
LIN {X 0,Y 559.206,Z 128.828,A -85,B 0,C 180,E1 -2874.23,E2 -2874.23} C_VEL
LIN {X 0,Y 559.251,Z 128.826,A -85,B 0,C 180,E1 -2877.84,E2 -2877.84} C_VEL
LIN {X 0,Y 559.258,Z 128.823,A -85,B 0,C 180,E1 -2880,E2 -2880} C_VEL
LIN {X 0,Y 559.208,Z 128.822,A -85,B 0,C 180,E1 -2882.882,E2 -2882.882} C_VEL
LIN {X 0,Y 559.208,Z 128.831,A -85,B 0,C 180,E1 -2885.771,E2 -2885.771} C_VEL
LIN {X 0,Y 559.155,Z 128.829,A -85,B 0,C 180,E1 -2888.675,E2 -2888.675} C_VEL
LIN {X 0,Y 559.201,Z 128.832,A -85,B 0,C 180,E1 -2891.601,E2 -2891.601} C_VEL
LIN {X 0,Y 559.159,Z 128.828,A -85,B 0,C 180,E1 -2894.576,E2 -2894.576} C_VEL
LIN {X 0,Y 559.118,Z 128.84,A -85,B 0,C 180,E1 -2897.559,E2 -2897.559} C_VEL
LIN {X 0,Y 559.152,Z 128.832,A -85,B 0,C 180,E1 -2899.838,E2 -2899.838} C_VEL
LIN {X 0,Y 559.108,Z 128.835,A -85,B 0,C 180,E1 -2902.155,E2 -2902.155} C_VEL
LIN {X 0,Y 559.144,Z 128.84,A -85,B 0,C 180,E1 -2905.178,E2 -2905.178} C_VEL
LIN {X 0,Y 559.107,Z 128.837,A -85,B 0,C 180,E1 -2907.717,E2 -2907.717} C_VEL
LIN {X 0,Y 559.102,Z 128.835,A -85,B 0,C 180,E1 -2910.186,E2 -2910.186} C_VEL
LIN {X 0,Y 559.152,Z 128.834,A -85,B 0,C 180,E1 -2912.716,E2 -2912.716} C_VEL
LIN {X 0,Y 559.121,Z 128.837,A -85,B 0,C 180,E1 -2915.325,E2 -2915.325} C_VEL
LIN {X 0,Y 559.13,Z 128.832,A -85,B 0,C 180,E1 -2918.018,E2 -2918.018} C_VEL
LIN {X 0,Y 559.157,Z 128.839,A -85,B 0,C 180,E1 -2920.813,E2 -2920.813} C_VEL
LIN {X 0,Y 559.111,Z 128.834,A -85,B 0,C 180,E1 -2923.737,E2 -2923.737} C_VEL
LIN {X 0,Y 559.111,Z 128.838,A -85,B 0,C 180,E1 -2926.263,E2 -2926.263} C_VEL
LIN {X 0,Y 559.156,Z 128.83,A -85,B 0,C 180,E1 -2929.187,E2 -2929.187} C_VEL
LIN {X 0,Y 559.127,Z 128.834,A -85,B 0,C 180,E1 -2931.981,E2 -2931.981} C_VEL
LIN {X 0,Y 559.126,Z 128.837,A -85,B 0,C 180,E1 -2934.789,E2 -2934.789} C_VEL
LIN {X 0,Y 559.152,Z 128.829,A -85,B 0,C 180,E1 -2937.366,E2 -2937.366} C_VEL
LIN {X 0,Y 559.122,Z 128.84,A -85,B 0,C 180,E1 -2940.148,E2 -2940.148} C_VEL
LIN {X 0,Y 559.127,Z 128.835,A -85,B 0,C 180,E1 -2943.182,E2 -2943.182} C_VEL
LIN {X 0,Y 559.159,Z 128.838,A -85,B 0,C 180,E1 -2946.259,E2 -2946.259} C_VEL
LIN {X 0,Y 560.056,Z 134.288,A -85,B 0,C 180,E1 -2947.107,E2 -2947.107} C_VEL
LIN {X 0,Y 559.888,Z 152.711,A -85,B 0,C 180,E1 -2949.806,E2 -2949.806} C_VEL
LIN {X 0,Y 559.569,Z 174.389,A -85,B 0,C 180,E1 -2952.931,E2 -2952.931} C_VEL
LIN {X 0,Y 559.375,Z 194.493,A -85,B 0,C 180,E1 -2955.795,E2 -2955.795} C_VEL
LIN {X 0,Y 560.255,Z 202.158,A -85,B 0,C 180,E1 -2955.933,E2 -2955.933} C_VEL
LIN {X 0,Y 560.04,Z 302.933,A -85,B 0,C 180,E1 -2957.245,E2 -2957.245} C_VEL
LIN {X 0,Y 559.914,Z 316.209,A -85,B 0,C 180,E1 -2957.564,E2 -2957.564} C_VEL
LIN {X 0,Y 559.792,Z 328.371,A -85,B 0,C 180,E1 -2957.999,E2 -2957.999} C_VEL
LIN {X 0,Y 559.644,Z 340.052,A -85,B 0,C 180,E1 -2958.56,E2 -2958.56} C_VEL
LIN {X 0,Y 559.458,Z 352.19,A -85,B 0,C 180,E1 -2959.322,E2 -2959.322} C_VEL
LIN {X 0,Y 559.306,Z 362.603,A -85,B 0,C 180,E1 -2960.142,E2 -2960.142} C_VEL
LIN {X 0,Y 559.162,Z 371.111,A -85,B 0,C 180,E1 -2960.961,E2 -2960.961} C_VEL
LIN {X 0,Y 559.05,Z 378.959,A -85,B 0,C 180,E1 -2961.869,E2 -2961.869} C_VEL
LIN {X 0,Y 558.944,Z 386.622,A -85,B 0,C 180,E1 -2962.958,E2 -2962.958} C_VEL
LIN {X 0,Y 558.936,Z 393.679,A -85,B 0,C 180,E1 -2964.227,E2 -2964.227} C_VEL
LIN {X 0,Y 558.826,Z 398.372,A -85,B 0,C 180,E1 -2965.311,E2 -2965.311} C_VEL
LIN {X 0,Y 558.836,Z 401.958,A -85,B 0,C 180,E1 -2966.395,E2 -2966.395} C_VEL
LIN {X 0,Y 558.799,Z 403.807,A -85,B 0,C 180,E1 -2967.116,E2 -2967.116} C_VEL
LIN {X 0,Y 558.745,Z 406.183,A -85,B 0,C 180,E1 -2968.558,E2 -2968.558} C_VEL
LIN {X 0,Y 558.74,Z 407,A -85,B 0,C 180,E1 -2970,E2 -2970} C_VEL
LIN {X 0,Y 558.745,Z 406.184,A -85,B 0,C 180,E1 -2971.441,E2 -2971.441} C_VEL
LIN {X 0,Y 558.799,Z 403.81,A -85,B 0,C 180,E1 -2972.884,E2 -2972.884} C_VEL
LIN {X 0,Y 558.844,Z 400.896,A -85,B 0,C 180,E1 -2973.966,E2 -2973.966} C_VEL
LIN {X 0,Y 558.798,Z 396.949,A -85,B 0,C 180,E1 -2975.051,E2 -2975.051} C_VEL
LIN {X 0,Y 558.922,Z 391.868,A -85,B 0,C 180,E1 -2976.135,E2 -2976.135} C_VEL
LIN {X 0,Y 558.977,Z 385.467,A -85,B 0,C 180,E1 -2977.223,E2 -2977.223} C_VEL
LIN {X 0,Y 559.099,Z 377.478,A -85,B 0,C 180,E1 -2978.312,E2 -2978.312} C_VEL
LIN {X 0,Y 559.195,Z 369.334,A -85,B 0,C 180,E1 -2979.221,E2 -2979.221} C_VEL
LIN {X 0,Y 559.357,Z 359.398,A -85,B 0,C 180,E1 -2980.131,E2 -2980.131} C_VEL
LIN {X 0,Y 559.556,Z 348.397,A -85,B 0,C 180,E1 -2980.937,E2 -2980.937} C_VEL
LIN {X 0,Y 559.672,Z 336.457,A -85,B 0,C 180,E1 -2981.628,E2 -2981.628} C_VEL
LIN {X 0,Y 559.822,Z 324.976,A -85,B 0,C 180,E1 -2982.138,E2 -2982.138} C_VEL
LIN {X 0,Y 559.98,Z 312.174,A -85,B 0,C 180,E1 -2982.549,E2 -2982.549} C_VEL
LIN {X 0,Y 560.081,Z 298.594,A -85,B 0,C 180,E1 -2982.823,E2 -2982.823} C_VEL
LIN {X 0,Y 560.202,Z 200.159,A -85,B 0,C 180,E1 -2984.094,E2 -2984.094} C_VEL
LIN {X 0,Y 559.373,Z 194.474,A -85,B 0,C 180,E1 -2984.205,E2 -2984.205} C_VEL
LIN {X 0,Y 559.568,Z 174.348,A -85,B 0,C 180,E1 -2987.064,E2 -2987.064} C_VEL
LIN {X 0,Y 559.833,Z 153.892,A -85,B 0,C 180,E1 -2990.004,E2 -2990.004} C_VEL
LIN {X 0,Y 560.048,Z 135.413,A -85,B 0,C 180,E1 -2992.698,E2 -2992.698} C_VEL
LIN {X 0,Y 559.149,Z 128.839,A -85,B 0,C 180,E1 -2993.717,E2 -2993.717} C_VEL
LIN {X 0,Y 559.159,Z 128.835,A -85,B 0,C 180,E1 -2996.098,E2 -2996.098} C_VEL
LIN {X 0,Y 559.111,Z 128.842,A -85,B 0,C 180,E1 -2999.356,E2 -2999.356} C_VEL
LIN {X 0,Y 559.157,Z 128.834,A -85,B 0,C 180,E1 -3001.863,E2 -3001.863} C_VEL
LIN {X 0,Y 559.129,Z 128.832,A -85,B 0,C 180,E1 -3004.446,E2 -3004.446} C_VEL
LIN {X 0,Y 559.13,Z 128.838,A -85,B 0,C 180,E1 -3007.109,E2 -3007.109} C_VEL
LIN {X 0,Y 559.151,Z 128.83,A -85,B 0,C 180,E1 -3009.94,E2 -3009.94} C_VEL
LIN {X 0,Y 559.124,Z 128.842,A -85,B 0,C 180,E1 -3013.194,E2 -3013.194} C_VEL
LIN {X 0,Y 559.125,Z 128.834,A -85,B 0,C 180,E1 -3015.764,E2 -3015.764} C_VEL
LIN {X 0,Y 559.098,Z 128.837,A -85,B 0,C 180,E1 -3018.223,E2 -3018.223} C_VEL
LIN {X 0,Y 559.127,Z 128.839,A -85,B 0,C 180,E1 -3021.062,E2 -3021.062} C_VEL
LIN {X 0,Y 559.109,Z 128.835,A -85,B 0,C 180,E1 -3023.787,E2 -3023.787} C_VEL
LIN {X 0,Y 559.106,Z 128.839,A -85,B 0,C 180,E1 -3026.421,E2 -3026.421} C_VEL
LIN {X 0,Y 559.136,Z 128.835,A -85,B 0,C 180,E1 -3028.979,E2 -3028.979} C_VEL
LIN {X 0,Y 559.104,Z 128.835,A -85,B 0,C 180,E1 -3031.632,E2 -3031.632} C_VEL
LIN {X 0,Y 559.143,Z 128.831,A -85,B 0,C 180,E1 -3033.901,E2 -3033.901} C_VEL
LIN {X 0,Y 559.093,Z 128.836,A -85,B 0,C 180,E1 -3037.065,E2 -3037.065} C_VEL
LIN {X 0,Y 559.109,Z 128.835,A -85,B 0,C 180,E1 -3039.392,E2 -3039.392} C_VEL
LIN {X 0,Y 559.113,Z 128.84,A -85,B 0,C 180,E1 -3042.441,E2 -3042.441} C_VEL
LIN {X 0,Y 559.156,Z 128.83,A -85,B 0,C 180,E1 -3045.441,E2 -3045.441} C_VEL
LIN {X 0,Y 559.159,Z 128.832,A -85,B 0,C 180,E1 -3048.398,E2 -3048.398} C_VEL
LIN {X 0,Y 559.163,Z 128.829,A -85,B 0,C 180,E1 -3051.325,E2 -3051.325} C_VEL
LIN {X 0,Y 559.213,Z 128.825,A -85,B 0,C 180,E1 -3054.229,E2 -3054.229} C_VEL
LIN {X 0,Y 559.253,Z 128.824,A -85,B 0,C 180,E1 -3057.839,E2 -3057.839} C_VEL
LIN {X 0,Y 559.259,Z 128.819,A -85,B 0,C 180,E1 -3060,E2 -3060} C_VEL
LIN {X 0,Y 559.224,Z 128.821,A -85,B 0,C 180,E1 -3062.881,E2 -3062.881} C_VEL
LIN {X 0,Y 559.221,Z 128.824,A -85,B 0,C 180,E1 -3065.77,E2 -3065.77} C_VEL
LIN {X 0,Y 559.167,Z 128.829,A -85,B 0,C 180,E1 -3068.674,E2 -3068.674} C_VEL
LIN {X 0,Y 559.207,Z 128.827,A -85,B 0,C 180,E1 -3071.6,E2 -3071.6} C_VEL
LIN {X 0,Y 559.183,Z 128.826,A -85,B 0,C 180,E1 -3074.587,E2 -3074.587} C_VEL
LIN {X 0,Y 559.135,Z 128.833,A -85,B 0,C 180,E1 -3077.557,E2 -3077.557} C_VEL
LIN {X 0,Y 559.166,Z 128.828,A -85,B 0,C 180,E1 -3079.837,E2 -3079.837} C_VEL
LIN {X 0,Y 559.136,Z 128.831,A -85,B 0,C 180,E1 -3082.153,E2 -3082.153} C_VEL
LIN {X 0,Y 559.144,Z 128.835,A -85,B 0,C 180,E1 -3085.178,E2 -3085.178} C_VEL
LIN {X 0,Y 559.148,Z 128.83,A -85,B 0,C 180,E1 -3087.713,E2 -3087.713} C_VEL
LIN {X 0,Y 559.136,Z 128.833,A -85,B 0,C 180,E1 -3090.581,E2 -3090.581} C_VEL
LIN {X 0,Y 558.473,Z 128.918,A -85,B 0,C 180,E1 -3091.182,E2 -3091.182} C_VEL
LIN {X 0,Y 555.611,Z 129.274,A -85,B 0,C 180,E1 -3092.158,E2 -3092.158} C_VEL
LIN {X 0,Y 553.196,Z 129.576,A -85,B 0,C 180,E1 -3092.944,E2 -3092.944} C_VEL
LIN {X 0,Y 552.168,Z 129.7,A -85,B 0,C 180,E1 -3093.551,E2 -3093.551} C_VEL
LIN {X 0,Y 552.09,Z 129.71,A -85,B 0,C 180,E1 -3093.756,E2 -3093.756} C_VEL
LIN {X 0,Y 552.105,Z 129.714,A -85,B 0,C 180,E1 -3096.747,E2 -3096.747} C_VEL
LIN {X 0,Y 552.129,Z 129.706,A -85,B 0,C 180,E1 -3099.527,E2 -3099.527} C_VEL
LIN {X 0,Y 552.13,Z 129.714,A -85,B 0,C 180,E1 -3102.425,E2 -3102.425} C_VEL
LIN {X 0,Y 552.097,Z 129.712,A -85,B 0,C 180,E1 -3105.562,E2 -3105.562} C_VEL
LIN {X 0,Y 552.136,Z 129.708,A -85,B 0,C 180,E1 -3108.676,E2 -3108.676} C_VEL
LIN {X 0,Y 552.192,Z 129.763,A -85,B 0,C 180,E1 -3110.728,E2 -3110.728} C_VEL
LIN {X 0,Y 552.477,Z 135.544,A -85,B 0,C 180,E1 -3111.793,E2 -3111.793} C_VEL
LIN {X 0,Y 552.346,Z 148.613,A -85,B 0,C 180,E1 -3114.176,E2 -3114.176} C_VEL
LIN {X 0,Y 552.203,Z 156.815,A -85,B 0,C 180,E1 -3115.691,E2 -3115.691} C_VEL
LIN {X 0,Y 553.463,Z 164.99,A -85,B 0,C 180,E1 -3115.832,E2 -3115.832} C_VEL
LIN {X 0,Y 553.093,Z 263.773,A -85,B 0,C 180,E1 -3117.138,E2 -3117.138} C_VEL
LIN {X 0,Y 553.012,Z 277.124,A -85,B 0,C 180,E1 -3117.47,E2 -3117.47} C_VEL
LIN {X 0,Y 552.827,Z 289.581,A -85,B 0,C 180,E1 -3117.929,E2 -3117.929} C_VEL
LIN {X 0,Y 552.618,Z 301.293,A -85,B 0,C 180,E1 -3118.514,E2 -3118.514} C_VEL
LIN {X 0,Y 552.433,Z 313.475,A -85,B 0,C 180,E1 -3119.305,E2 -3119.305} C_VEL
LIN {X 0,Y 552.288,Z 323.021,A -85,B 0,C 180,E1 -3120.08,E2 -3120.08} C_VEL
LIN {X 0,Y 552.129,Z 331.025,A -85,B 0,C 180,E1 -3120.864,E2 -3120.864} C_VEL
LIN {X 0,Y 551.993,Z 339.718,A -85,B 0,C 180,E1 -3121.895,E2 -3121.895} C_VEL
LIN {X 0,Y 551.857,Z 347.563,A -85,B 0,C 180,E1 -3123.057,E2 -3123.057} C_VEL
LIN {X 0,Y 551.796,Z 354.391,A -85,B 0,C 180,E1 -3124.339,E2 -3124.339} C_VEL
LIN {X 0,Y 551.733,Z 359.278,A -85,B 0,C 180,E1 -3125.544,E2 -3125.544} C_VEL
LIN {X 0,Y 551.705,Z 362.88,A -85,B 0,C 180,E1 -3126.74,E2 -3126.74} C_VEL
LIN {X 0,Y 551.659,Z 364.622,A -85,B 0,C 180,E1 -3127.53,E2 -3127.53} C_VEL
LIN {X 0,Y 551.669,Z 366.015,A -85,B 0,C 180,E1 -3128.431,E2 -3128.431} C_VEL
LIN {X 0,Y 551.639,Z 366.97,A -85,B 0,C 180,E1 -3129.88,E2 -3129.88} C_VEL
LIN {X 0,Y 551.679,Z 366.86,A -85,B 0,C 180,E1 -3130.657,E2 -3130.657} C_VEL
LIN {X 0,Y 551.643,Z 366.266,A -85,B 0,C 180,E1 -3131.428,E2 -3131.428} C_VEL
LIN {X 0,Y 551.678,Z 364.08,A -85,B 0,C 180,E1 -3132.831,E2 -3132.831} C_VEL
LIN {X 0,Y 551.727,Z 360.764,A -85,B 0,C 180,E1 -3134.105,E2 -3134.105} C_VEL
LIN {X 0,Y 551.786,Z 355.652,A -85,B 0,C 180,E1 -3135.464,E2 -3135.464} C_VEL
LIN {X 0,Y 551.814,Z 349.263,A -85,B 0,C 180,E1 -3136.747,E2 -3136.747} C_VEL
LIN {X 0,Y 551.965,Z 342.073,A -85,B 0,C 180,E1 -3137.872,E2 -3137.872} C_VEL
LIN {X 0,Y 552.085,Z 333.143,A -85,B 0,C 180,E1 -3138.992,E2 -3138.992} C_VEL
LIN {X 0,Y 552.248,Z 323.992,A -85,B 0,C 180,E1 -3139.922,E2 -3139.922} C_VEL
LIN {X 0,Y 552.435,Z 313.844,A -85,B 0,C 180,E1 -3140.758,E2 -3140.758} C_VEL
LIN {X 0,Y 552.653,Z 302.577,A -85,B 0,C 180,E1 -3141.499,E2 -3141.499} C_VEL
LIN {X 0,Y 552.813,Z 290.662,A -85,B 0,C 180,E1 -3142.113,E2 -3142.113} C_VEL
LIN {X 0,Y 552.95,Z 278.65,A -85,B 0,C 180,E1 -3142.574,E2 -3142.574} C_VEL
LIN {X 0,Y 553.102,Z 265.302,A -85,B 0,C 180,E1 -3142.92,E2 -3142.92} C_VEL
LIN {X 0,Y 553.189,Z 243.644,A -85,B 0,C 180,E1 -3143.234,E2 -3143.234} C_VEL
LIN {X 0,Y 553.318,Z 163.346,A -85,B 0,C 180,E1 -3144.282,E2 -3144.282} C_VEL
LIN {X 0,Y 552.232,Z 156.765,A -85,B 0,C 180,E1 -3144.408,E2 -3144.408} C_VEL
LIN {X 0,Y 552.398,Z 140.327,A -85,B 0,C 180,E1 -3147.448,E2 -3147.448} C_VEL
LIN {X 0,Y 552.443,Z 132.453,A -85,B 0,C 180,E1 -3148.907,E2 -3148.907} C_VEL
LIN {X 0,Y 552.078,Z 129.718,A -85,B 0,C 180,E1 -3149.453,E2 -3149.453} C_VEL
LIN {X 0,Y 552.109,Z 129.711,A -85,B 0,C 180,E1 -3151.459,E2 -3151.459} C_VEL
LIN {X 0,Y 552.169,Z 129.701,A -85,B 0,C 180,E1 -3152.918,E2 -3152.918} C_VEL
LIN {X 0,Y 552.169,Z 129.707,A -85,B 0,C 180,E1 -3155.844,E2 -3155.844} C_VEL
LIN {X 0,Y 552.118,Z 129.705,A -85,B 0,C 180,E1 -3158.787,E2 -3158.787} C_VEL
LIN {X 0,Y 552.093,Z 129.718,A -85,B 0,C 180,E1 -3161.752,E2 -3161.752} C_VEL
LIN {X 0,Y 552.113,Z 129.706,A -85,B 0,C 180,E1 -3164.749,E2 -3164.749} C_VEL
LIN {X 0,Y 552.064,Z 129.719,A -85,B 0,C 180,E1 -3167.79,E2 -3167.79} C_VEL
LIN {X 0,Y 552.042,Z 129.717,A -85,B 0,C 180,E1 -3170.105,E2 -3170.105} C_VEL
LIN {X 0,Y 552.036,Z 129.716,A -85,B 0,C 180,E1 -3172.454,E2 -3172.454} C_VEL
LIN {X 0,Y 552.06,Z 129.72,A -85,B 0,C 180,E1 -3175.33,E2 -3175.33} C_VEL
LIN {X 0,Y 552.043,Z 129.715,A -85,B 0,C 180,E1 -3178.102,E2 -3178.102} C_VEL
LIN {X 0,Y 552.063,Z 129.713,A -85,B 0,C 180,E1 -3180.612,E2 -3180.612} C_VEL
LIN {X 0,Y 552.085,Z 129.718,A -85,B 0,C 180,E1 -3183.188,E2 -3183.188} C_VEL
LIN {X 0,Y 552.06,Z 129.714,A -85,B 0,C 180,E1 -3185.846,E2 -3185.846} C_VEL
LIN {X 0,Y 552.081,Z 129.712,A -85,B 0,C 180,E1 -3188.592,E2 -3188.592} C_VEL
LIN {X 0,Y 552.051,Z 129.717,A -85,B 0,C 180,E1 -3191.453,E2 -3191.453} C_VEL
LIN {X 0,Y 552.073,Z 129.714,A -85,B 0,C 180,E1 -3194.53,E2 -3194.53} C_VEL
LIN {X 0,Y 552.078,Z 129.711,A -85,B 0,C 180,E1 -3197.591,E2 -3197.591} C_VEL
LIN {X 0,Y 552.091,Z 129.713,A -85,B 0,C 180,E1 -3200.47,E2 -3200.47} C_VEL
LIN {X 0,Y 552.069,Z 129.713,A -85,B 0,C 180,E1 -3203.323,E2 -3203.323} C_VEL
LIN {X 0,Y 552.083,Z 129.71,A -85,B 0,C 180,E1 -3205.937,E2 -3205.937} C_VEL
LIN {X 0,Y 552.08,Z 129.718,A -85,B 0,C 180,E1 -3208.539,E2 -3208.539} C_VEL
LIN {X 0,Y 552.071,Z 129.711,A -85,B 0,C 180,E1 -3211.449,E2 -3211.449} C_VEL
LIN {X 0,Y 552.071,Z 129.719,A -85,B 0,C 180,E1 -3214.353,E2 -3214.353} C_VEL
LIN {X 0,Y 552.046,Z 129.719,A -85,B 0,C 180,E1 -3216.756,E2 -3216.756} C_VEL
LIN {X 0,Y 552.068,Z 129.712,A -85,B 0,C 180,E1 -3219.118,E2 -3219.118} C_VEL
LIN {X 0,Y 552.048,Z 129.714,A -85,B 0,C 180,E1 -3221.442,E2 -3221.442} C_VEL
LIN {X 0,Y 552.071,Z 129.714,A -85,B 0,C 180,E1 -3223.736,E2 -3223.736} C_VEL
LIN {X 0,Y 552.106,Z 129.714,A -85,B 0,C 180,E1 -3226.004,E2 -3226.004} C_VEL
LIN {X 0,Y 552.129,Z 129.704,A -85,B 0,C 180,E1 -3228.993,E2 -3228.993} C_VEL
LIN {X 0,Y 552.112,Z 129.714,A -85,B 0,C 180,E1 -3231.951,E2 -3231.951} C_VEL
LIN {X 0,Y 552.205,Z 129.695,A -85,B 0,C 180,E1 -3234.889,E2 -3234.889} C_VEL
LIN {X 0,Y 552.222,Z 129.701,A -85,B 0,C 180,E1 -3237.812,E2 -3237.812} C_VEL
LIN {X 0,Y 552.226,Z 129.699,A -85,B 0,C 180,E1 -3240,E2 -3240} C_VEL
LIN {X 0,Y 552.176,Z 129.698,A -85,B 0,C 180,E1 -3242.919,E2 -3242.919} C_VEL
LIN {X 0,Y 552.178,Z 129.705,A -85,B 0,C 180,E1 -3245.844,E2 -3245.844} C_VEL
LIN {X 0,Y 552.128,Z 129.704,A -85,B 0,C 180,E1 -3248.787,E2 -3248.787} C_VEL
LIN {X 0,Y 552.154,Z 129.707,A -85,B 0,C 180,E1 -3251.751,E2 -3251.751} C_VEL
LIN {X 0,Y 552.125,Z 129.705,A -85,B 0,C 180,E1 -3254.749,E2 -3254.749} C_VEL
LIN {X 0,Y 552.082,Z 129.713,A -85,B 0,C 180,E1 -3257.79,E2 -3257.79} C_VEL
LIN {X 0,Y 552.104,Z 129.708,A -85,B 0,C 180,E1 -3260.103,E2 -3260.103} C_VEL
LIN {X 0,Y 552.048,Z 129.714,A -85,B 0,C 180,E1 -3262.453,E2 -3262.453} C_VEL
LIN {X 0,Y 552.087,Z 129.717,A -85,B 0,C 180,E1 -3265.334,E2 -3265.334} C_VEL
LIN {X 0,Y 552.054,Z 129.713,A -85,B 0,C 180,E1 -3268.102,E2 -3268.102} C_VEL
LIN {X 0,Y 552.078,Z 129.713,A -85,B 0,C 180,E1 -3270.611,E2 -3270.611} C_VEL
LIN {X 0,Y 552.108,Z 129.713,A -85,B 0,C 180,E1 -3273.187,E2 -3273.187} C_VEL
LIN {X 0,Y 552.075,Z 129.711,A -85,B 0,C 180,E1 -3275.845,E2 -3275.845} C_VEL
LIN {X 0,Y 552.117,Z 129.711,A -85,B 0,C 180,E1 -3278.589,E2 -3278.589} C_VEL
LIN {X 0,Y 552.077,Z 129.712,A -85,B 0,C 180,E1 -3281.45,E2 -3281.45} C_VEL
LIN {X 0,Y 552.079,Z 129.717,A -85,B 0,C 180,E1 -3284.529,E2 -3284.529} C_VEL
LIN {X 0,Y 552.09,Z 129.709,A -85,B 0,C 180,E1 -3287.59,E2 -3287.59} C_VEL
LIN {X 0,Y 552.128,Z 129.712,A -85,B 0,C 180,E1 -3290.472,E2 -3290.472} C_VEL
LIN {X 0,Y 552.101,Z 129.708,A -85,B 0,C 180,E1 -3293.318,E2 -3293.318} C_VEL
LIN {X 0,Y 552.101,Z 129.71,A -85,B 0,C 180,E1 -3295.937,E2 -3295.937} C_VEL
LIN {X 0,Y 552.124,Z 129.713,A -85,B 0,C 180,E1 -3298.54,E2 -3298.54} C_VEL
LIN {X 0,Y 552.083,Z 129.711,A -85,B 0,C 180,E1 -3301.447,E2 -3301.447} C_VEL
LIN {X 0,Y 552.086,Z 129.72,A -85,B 0,C 180,E1 -3304.353,E2 -3304.353} C_VEL
LIN {X 0,Y 552.103,Z 129.786,A -85,B 0,C 180,E1 -3306.116,E2 -3306.116} C_VEL
LIN {X 0,Y 553.082,Z 135.365,A -85,B 0,C 180,E1 -3306.999,E2 -3306.999} C_VEL
LIN {X 0,Y 552.915,Z 149.832,A -85,B 0,C 180,E1 -3309.151,E2 -3309.151} C_VEL
LIN {X 0,Y 552.646,Z 169.531,A -85,B 0,C 180,E1 -3312.038,E2 -3312.038} C_VEL
LIN {X 0,Y 552.386,Z 188.003,A -85,B 0,C 180,E1 -3314.711,E2 -3314.711} C_VEL
LIN {X 0,Y 552.36,Z 194.362,A -85,B 0,C 180,E1 -3315.627,E2 -3315.627} C_VEL
LIN {X 0,Y 553.359,Z 202.397,A -85,B 0,C 180,E1 -3315.762,E2 -3315.762} C_VEL
LIN {X 0,Y 553.131,Z 302.621,A -85,B 0,C 180,E1 -3317.083,E2 -3317.083} C_VEL
LIN {X 0,Y 552.979,Z 315.939,A -85,B 0,C 180,E1 -3317.406,E2 -3317.406} C_VEL
LIN {X 0,Y 552.847,Z 328.135,A -85,B 0,C 180,E1 -3317.845,E2 -3317.845} C_VEL
LIN {X 0,Y 552.657,Z 338.967,A -85,B 0,C 180,E1 -3318.365,E2 -3318.365} C_VEL
LIN {X 0,Y 552.482,Z 350.761,A -85,B 0,C 180,E1 -3319.092,E2 -3319.092} C_VEL
LIN {X 0,Y 552.298,Z 361.448,A -85,B 0,C 180,E1 -3319.923,E2 -3319.923} C_VEL
LIN {X 0,Y 552.132,Z 371.077,A -85,B 0,C 180,E1 -3320.845,E2 -3320.845} C_VEL
LIN {X 0,Y 552.014,Z 378.959,A -85,B 0,C 180,E1 -3321.765,E2 -3321.765} C_VEL
LIN {X 0,Y 551.89,Z 386.62,A -85,B 0,C 180,E1 -3322.868,E2 -3322.868} C_VEL
LIN {X 0,Y 551.867,Z 393.678,A -85,B 0,C 180,E1 -3324.152,E2 -3324.152} C_VEL
LIN {X 0,Y 551.725,Z 398.372,A -85,B 0,C 180,E1 -3325.25,E2 -3325.25} C_VEL
LIN {X 0,Y 551.75,Z 401.957,A -85,B 0,C 180,E1 -3326.348,E2 -3326.348} C_VEL
LIN {X 0,Y 551.724,Z 403.806,A -85,B 0,C 180,E1 -3327.079,E2 -3327.079} C_VEL
LIN {X 0,Y 551.645,Z 406.182,A -85,B 0,C 180,E1 -3328.54,E2 -3328.54} C_VEL
LIN {X 0,Y 551.64,Z 407,A -85,B 0,C 180,E1 -3330,E2 -3330} C_VEL
LIN {X 0,Y 551.645,Z 406.184,A -85,B 0,C 180,E1 -3331.46,E2 -3331.46} C_VEL
LIN {X 0,Y 551.724,Z 403.81,A -85,B 0,C 180,E1 -3332.921,E2 -3332.921} C_VEL
LIN {X 0,Y 551.764,Z 400.895,A -85,B 0,C 180,E1 -3334.017,E2 -3334.017} C_VEL
LIN {X 0,Y 551.724,Z 396.948,A -85,B 0,C 180,E1 -3335.116,E2 -3335.116} C_VEL
LIN {X 0,Y 551.803,Z 391.19,A -85,B 0,C 180,E1 -3336.341,E2 -3336.341} C_VEL
LIN {X 0,Y 551.927,Z 384.235,A -85,B 0,C 180,E1 -3337.5,E2 -3337.5} C_VEL
LIN {X 0,Y 552.082,Z 375.987,A -85,B 0,C 180,E1 -3338.602,E2 -3338.602} C_VEL
LIN {X 0,Y 552.201,Z 367.485,A -85,B 0,C 180,E1 -3339.524,E2 -3339.524} C_VEL
LIN {X 0,Y 552.412,Z 356.98,A -85,B 0,C 180,E1 -3340.445,E2 -3340.445} C_VEL
LIN {X 0,Y 552.575,Z 346.122,A -85,B 0,C 180,E1 -3341.214,E2 -3341.214} C_VEL
LIN {X 0,Y 552.752,Z 335.194,A -85,B 0,C 180,E1 -3341.831,E2 -3341.831} C_VEL
LIN {X 0,Y 552.899,Z 323.505,A -85,B 0,C 180,E1 -3342.34,E2 -3342.34} C_VEL
LIN {X 0,Y 553.031,Z 310.037,A -85,B 0,C 180,E1 -3342.756,E2 -3342.756} C_VEL
LIN {X 0,Y 553.178,Z 296.72,A -85,B 0,C 180,E1 -3343.009,E2 -3343.009} C_VEL
LIN {X 0,Y 553.233,Z 200.336,A -85,B 0,C 180,E1 -3344.269,E2 -3344.269} C_VEL
LIN {X 0,Y 552.341,Z 194.178,A -85,B 0,C 180,E1 -3344.393,E2 -3344.393} C_VEL
LIN {X 0,Y 552.558,Z 173.7,A -85,B 0,C 180,E1 -3347.342,E2 -3347.342} C_VEL
LIN {X 0,Y 552.889,Z 153.612,A -85,B 0,C 180,E1 -3350.266,E2 -3350.266} C_VEL
LIN {X 0,Y 553.094,Z 136.449,A -85,B 0,C 180,E1 -3352.802,E2 -3352.802} C_VEL
LIN {X 0,Y 552.098,Z 129.717,A -85,B 0,C 180,E1 -3353.85,E2 -3353.85} C_VEL
LIN {X 0,Y 552.094,Z 129.712,A -85,B 0,C 180,E1 -3356.99,E2 -3356.99} C_VEL
LIN {X 0,Y 552.097,Z 129.714,A -85,B 0,C 180,E1 -3360.046,E2 -3360.046} C_VEL
LIN {X 0,Y 552.109,Z 129.709,A -85,B 0,C 180,E1 -3362.845,E2 -3362.845} C_VEL
LIN {X 0,Y 552.072,Z 129.715,A -85,B 0,C 180,E1 -3365.845,E2 -3365.845} C_VEL
LIN {X 0,Y 552.112,Z 129.708,A -85,B 0,C 180,E1 -3368.59,E2 -3368.59} C_VEL
LIN {X 0,Y 552.06,Z 129.719,A -85,B 0,C 180,E1 -3371.452,E2 -3371.452} C_VEL
LIN {X 0,Y 552.077,Z 129.712,A -85,B 0,C 180,E1 -3374.529,E2 -3374.529} C_VEL
LIN {X 0,Y 552.082,Z 129.713,A -85,B 0,C 180,E1 -3377.59,E2 -3377.59} C_VEL
LIN {X 0,Y 552.077,Z 129.714,A -85,B 0,C 180,E1 -3380.468,E2 -3380.468} C_VEL
LIN {X 0,Y 552.052,Z 129.717,A -85,B 0,C 180,E1 -3383.325,E2 -3383.325} C_VEL
LIN {X 0,Y 552.073,Z 129.71,A -85,B 0,C 180,E1 -3385.935,E2 -3385.935} C_VEL
LIN {X 0,Y 552.082,Z 129.718,A -85,B 0,C 180,E1 -3388.538,E2 -3388.538} C_VEL
LIN {X 0,Y 552.072,Z 129.711,A -85,B 0,C 180,E1 -3391.449,E2 -3391.449} C_VEL
LIN {X 0,Y 552.069,Z 129.717,A -85,B 0,C 180,E1 -3394.352,E2 -3394.352} C_VEL
LIN {X 0,Y 552.047,Z 129.716,A -85,B 0,C 180,E1 -3396.755,E2 -3396.755} C_VEL
LIN {X 0,Y 552.069,Z 129.712,A -85,B 0,C 180,E1 -3399.117,E2 -3399.117} C_VEL
LIN {X 0,Y 552.049,Z 129.714,A -85,B 0,C 180,E1 -3401.441,E2 -3401.441} C_VEL
LIN {X 0,Y 552.076,Z 129.713,A -85,B 0,C 180,E1 -3403.736,E2 -3403.736} C_VEL
LIN {X 0,Y 552.11,Z 129.715,A -85,B 0,C 180,E1 -3406.003,E2 -3406.003} C_VEL
LIN {X 0,Y 552.132,Z 129.704,A -85,B 0,C 180,E1 -3408.992,E2 -3408.992} C_VEL
LIN {X 0,Y 552.115,Z 129.713,A -85,B 0,C 180,E1 -3411.951,E2 -3411.951} C_VEL
LIN {X 0,Y 552.212,Z 129.694,A -85,B 0,C 180,E1 -3414.888,E2 -3414.888} C_VEL
LIN {X 0,Y 552.224,Z 129.7,A -85,B 0,C 180,E1 -3417.812,E2 -3417.812} C_VEL
LIN {X 0,Y 552.228,Z 129.695,A -85,B 0,C 180,E1 -3420,E2 -3420} C_VEL
LIN {X 0,Y 552.193,Z 129.697,A -85,B 0,C 180,E1 -3422.918,E2 -3422.918} C_VEL
LIN {X 0,Y 552.191,Z 129.699,A -85,B 0,C 180,E1 -3425.844,E2 -3425.844} C_VEL
LIN {X 0,Y 552.139,Z 129.705,A -85,B 0,C 180,E1 -3428.786,E2 -3428.786} C_VEL
LIN {X 0,Y 552.163,Z 129.703,A -85,B 0,C 180,E1 -3431.75,E2 -3431.75} C_VEL
LIN {X 0,Y 552.131,Z 129.706,A -85,B 0,C 180,E1 -3434.748,E2 -3434.748} C_VEL
LIN {X 0,Y 552.094,Z 129.709,A -85,B 0,C 180,E1 -3437.789,E2 -3437.789} C_VEL
LIN {X 0,Y 552.127,Z 129.705,A -85,B 0,C 180,E1 -3440.101,E2 -3440.101} C_VEL
LIN {X 0,Y 552.088,Z 129.711,A -85,B 0,C 180,E1 -3442.451,E2 -3442.451} C_VEL
LIN {X 0,Y 552.112,Z 129.707,A -85,B 0,C 180,E1 -3445.645,E2 -3445.645} C_VEL
LIN {X 0,Y 552.125,Z 129.712,A -85,B 0,C 180,E1 -3448.561,E2 -3448.561} C_VEL
LIN {X 0,Y 552.111,Z 129.707,A -85,B 0,C 180,E1 -3451.475,E2 -3451.475} C_VEL
LIN {X 0,Y 552.09,Z 129.71,A -85,B 0,C 180,E1 -3453.756,E2 -3453.756} C_VEL
LIN {X 0,Y 551.449,Z 129.796,A -85,B 0,C 180,E1 -3454.365,E2 -3454.365} C_VEL
LIN {X 0,Y 548.637,Z 130.148,A -85,B 0,C 180,E1 -3455.353,E2 -3455.353} C_VEL
LIN {X 0,Y 546.23,Z 130.448,A -85,B 0,C 180,E1 -3456.149,E2 -3456.149} C_VEL
LIN {X 0,Y 545.167,Z 130.579,A -85,B 0,C 180,E1 -3456.763,E2 -3456.763} C_VEL
LIN {X 0,Y 545.064,Z 130.588,A -85,B 0,C 180,E1 -3456.971,E2 -3456.971} C_VEL
LIN {X 0,Y 545.065,Z 130.592,A -85,B 0,C 180,E1 -3460.142,E2 -3460.142} C_VEL
LIN {X 0,Y 545.077,Z 130.586,A -85,B 0,C 180,E1 -3463.106,E2 -3463.106} C_VEL
LIN {X 0,Y 545.056,Z 130.594,A -85,B 0,C 180,E1 -3466.225,E2 -3466.225} C_VEL
LIN {X 0,Y 545.098,Z 130.584,A -85,B 0,C 180,E1 -3468.887,E2 -3468.887} C_VEL
LIN {X 0,Y 545.122,Z 130.614,A -85,B 0,C 180,E1 -3470.624,E2 -3470.624} C_VEL
LIN {X 0,Y 545.483,Z 135.647,A -85,B 0,C 180,E1 -3471.563,E2 -3471.563} C_VEL
LIN {X 0,Y 545.303,Z 150.436,A -85,B 0,C 180,E1 -3474.287,E2 -3474.287} C_VEL
LIN {X 0,Y 545.226,Z 157.173,A -85,B 0,C 180,E1 -3475.505,E2 -3475.505} C_VEL
LIN {X 0,Y 546.593,Z 165.886,A -85,B 0,C 180,E1 -3475.659,E2 -3475.659} C_VEL
LIN {X 0,Y 546.199,Z 263.849,A -85,B 0,C 180,E1 -3476.97,E2 -3476.97} C_VEL
LIN {X 0,Y 546.094,Z 276.89,A -85,B 0,C 180,E1 -3477.294,E2 -3477.294} C_VEL
LIN {X 0,Y 545.896,Z 289.502,A -85,B 0,C 180,E1 -3477.759,E2 -3477.759} C_VEL
LIN {X 0,Y 545.672,Z 301.156,A -85,B 0,C 180,E1 -3478.342,E2 -3478.342} C_VEL
LIN {X 0,Y 545.489,Z 312.556,A -85,B 0,C 180,E1 -3479.081,E2 -3479.081} C_VEL
LIN {X 0,Y 545.282,Z 323.042,A -85,B 0,C 180,E1 -3479.93,E2 -3479.93} C_VEL
LIN {X 0,Y 545.11,Z 332.099,A -85,B 0,C 180,E1 -3480.833,E2 -3480.833} C_VEL
LIN {X 0,Y 544.936,Z 340.903,A -85,B 0,C 180,E1 -3481.918,E2 -3481.918} C_VEL
LIN {X 0,Y 544.807,Z 347.337,A -85,B 0,C 180,E1 -3482.884,E2 -3482.884} C_VEL
LIN {X 0,Y 544.746,Z 353.291,A -85,B 0,C 180,E1 -3483.982,E2 -3483.982} C_VEL
LIN {X 0,Y 544.664,Z 358.515,A -85,B 0,C 180,E1 -3485.206,E2 -3485.206} C_VEL
LIN {X 0,Y 544.635,Z 362.396,A -85,B 0,C 180,E1 -3486.42,E2 -3486.42} C_VEL
LIN {X 0,Y 544.573,Z 364.291,A -85,B 0,C 180,E1 -3487.222,E2 -3487.222} C_VEL
LIN {X 0,Y 544.567,Z 366.101,A -85,B 0,C 180,E1 -3488.31,E2 -3488.31} C_VEL
LIN {X 0,Y 544.547,Z 367.098,A -85,B 0,C 180,E1 -3489.606,E2 -3489.606} C_VEL
LIN {X 0,Y 544.579,Z 367.114,A -85,B 0,C 180,E1 -3490.404,E2 -3490.404} C_VEL
LIN {X 0,Y 544.549,Z 366.719,A -85,B 0,C 180,E1 -3491.177,E2 -3491.177} C_VEL
LIN {X 0,Y 544.549,Z 365.855,A -85,B 0,C 180,E1 -3491.956,E2 -3491.956} C_VEL
LIN {X 0,Y 544.577,Z 364.525,A -85,B 0,C 180,E1 -3492.745,E2 -3492.745} C_VEL
LIN {X 0,Y 544.625,Z 361.756,A -85,B 0,C 180,E1 -3493.892,E2 -3493.892} C_VEL
LIN {X 0,Y 544.724,Z 357.889,A -85,B 0,C 180,E1 -3495.046,E2 -3495.046} C_VEL
LIN {X 0,Y 544.743,Z 352.879,A -85,B 0,C 180,E1 -3496.192,E2 -3496.192} C_VEL
LIN {X 0,Y 544.845,Z 346.562,A -85,B 0,C 180,E1 -3497.333,E2 -3497.333} C_VEL
LIN {X 0,Y 544.99,Z 339.065,A -85,B 0,C 180,E1 -3498.419,E2 -3498.419} C_VEL
LIN {X 0,Y 545.128,Z 330.607,A -85,B 0,C 180,E1 -3499.414,E2 -3499.414} C_VEL
LIN {X 0,Y 545.333,Z 320.791,A -85,B 0,C 180,E1 -3500.355,E2 -3500.355} C_VEL
LIN {X 0,Y 545.564,Z 309.842,A -85,B 0,C 180,E1 -3501.201,E2 -3501.201} C_VEL
LIN {X 0,Y 545.745,Z 299.14,A -85,B 0,C 180,E1 -3501.856,E2 -3501.856} C_VEL
LIN {X 0,Y 545.922,Z 287.36,A -85,B 0,C 180,E1 -3502.419,E2 -3502.419} C_VEL
LIN {X 0,Y 546.111,Z 274.12,A -85,B 0,C 180,E1 -3502.88,E2 -3502.88} C_VEL
LIN {X 0,Y 546.219,Z 260.785,A -85,B 0,C 180,E1 -3503.172,E2 -3503.172} C_VEL
LIN {X 0,Y 546.485,Z 164.353,A -85,B 0,C 180,E1 -3504.454,E2 -3504.454} C_VEL
LIN {X 0,Y 545.234,Z 156.991,A -85,B 0,C 180,E1 -3504.592,E2 -3504.592} C_VEL
LIN {X 0,Y 545.429,Z 139.842,A -85,B 0,C 180,E1 -3507.785,E2 -3507.785} C_VEL
LIN {X 0,Y 545.268,Z 131.973,A -85,B 0,C 180,E1 -3509.262,E2 -3509.262} C_VEL
LIN {X 0,Y 545.062,Z 130.593,A -85,B 0,C 180,E1 -3509.538,E2 -3509.538} C_VEL
LIN {X 0,Y 545.186,Z 130.578,A -85,B 0,C 180,E1 -3512.217,E2 -3512.217} C_VEL
LIN {X 0,Y 545.155,Z 130.573,A -85,B 0,C 180,E1 -3515.178,E2 -3515.178} C_VEL
LIN {X 0,Y 545.06,Z 130.59,A -85,B 0,C 180,E1 -3518.154,E2 -3518.154} C_VEL
LIN {X 0,Y 545.067,Z 130.585,A -85,B 0,C 180,E1 -3521.152,E2 -3521.152} C_VEL
LIN {X 0,Y 545.057,Z 130.588,A -85,B 0,C 180,E1 -3524.181,E2 -3524.181} C_VEL
LIN {X 0,Y 545.035,Z 130.593,A -85,B 0,C 180,E1 -3527.41,E2 -3527.41} C_VEL
LIN {X 0,Y 544.998,Z 130.593,A -85,B 0,C 180,E1 -3530.376,E2 -3530.376} C_VEL
LIN {X 0,Y 544.982,Z 130.595,A -85,B 0,C 180,E1 -3532.761,E2 -3532.761} C_VEL
LIN {X 0,Y 545.012,Z 130.6,A -85,B 0,C 180,E1 -3535.491,E2 -3535.491} C_VEL
LIN {X 0,Y 544.992,Z 130.598,A -85,B 0,C 180,E1 -3537.661,E2 -3537.661} C_VEL
LIN {X 0,Y 545.016,Z 130.59,A -85,B 0,C 180,E1 -3540.236,E2 -3540.236} C_VEL
LIN {X 0,Y 545.054,Z 130.592,A -85,B 0,C 180,E1 -3543.059,E2 -3543.059} C_VEL
LIN {X 0,Y 545.01,Z 130.593,A -85,B 0,C 180,E1 -3545.67,E2 -3545.67} C_VEL
LIN {X 0,Y 545.022,Z 130.589,A -85,B 0,C 180,E1 -3548.24,E2 -3548.24} C_VEL
LIN {X 0,Y 545.001,Z 130.6,A -85,B 0,C 180,E1 -3551.123,E2 -3551.123} C_VEL
LIN {X 0,Y 545.028,Z 130.589,A -85,B 0,C 180,E1 -3554.133,E2 -3554.133} C_VEL
LIN {X 0,Y 545.015,Z 130.6,A -85,B 0,C 180,E1 -3556.888,E2 -3556.888} C_VEL
LIN {X 0,Y 545.031,Z 130.588,A -85,B 0,C 180,E1 -3559.855,E2 -3559.855} C_VEL
LIN {X 0,Y 545.017,Z 130.598,A -85,B 0,C 180,E1 -3562.695,E2 -3562.695} C_VEL
LIN {X 0,Y 545.045,Z 130.587,A -85,B 0,C 180,E1 -3565.614,E2 -3565.614} C_VEL
LIN {X 0,Y 545.044,Z 130.591,A -85,B 0,C 180,E1 -3568.325,E2 -3568.325} C_VEL
LIN {X 0,Y 545.032,Z 130.588,A -85,B 0,C 180,E1 -3571.504,E2 -3571.504} C_VEL
LIN {X 0,Y 545.035,Z 130.59,A -85,B 0,C 180,E1 -3573.998,E2 -3573.998} C_VEL
LIN {X 0,Y 545.049,Z 130.596,A -85,B 0,C 180,E1 -3576.44,E2 -3576.44} C_VEL
LIN {X 0,Y 545.018,Z 130.593,A -85,B 0,C 180,E1 -3578.835,E2 -3578.835} C_VEL
LIN {X 0,Y 545.004,Z 130.592,A -85,B 0,C 180,E1 -3581.193,E2 -3581.193} C_VEL
LIN {X 0,Y 545.022,Z 130.59,A -85,B 0,C 180,E1 -3583.52,E2 -3583.52} C_VEL
LIN {X 0,Y 545.066,Z 130.588,A -85,B 0,C 180,E1 -3585.82,E2 -3585.82} C_VEL
LIN {X 0,Y 545.075,Z 130.583,A -85,B 0,C 180,E1 -3588.849,E2 -3588.849} C_VEL
LIN {X 0,Y 545.069,Z 130.59,A -85,B 0,C 180,E1 -3591.847,E2 -3591.847} C_VEL
LIN {X 0,Y 545.163,Z 130.572,A -85,B 0,C 180,E1 -3594.823,E2 -3594.823} C_VEL
LIN {X 0,Y 545.193,Z 130.576,A -85,B 0,C 180,E1 -3597.784,E2 -3597.784} C_VEL
LIN {X 0,Y 545.195,Z 130.575,A -85,B 0,C 180,E1 -3600,E2 -3600} C_VEL
LIN {X 0,Y 545.145,Z 130.574,A -85,B 0,C 180,E1 -3602.956,E2 -3602.956} C_VEL
LIN {X 0,Y 545.126,Z 130.582,A -85,B 0,C 180,E1 -3605.92,E2 -3605.92} C_VEL
LIN {X 0,Y 545.072,Z 130.584,A -85,B 0,C 180,E1 -3608.901,E2 -3608.901} C_VEL
LIN {X 0,Y 545.096,Z 130.584,A -85,B 0,C 180,E1 -3611.905,E2 -3611.905} C_VEL
LIN {X 0,Y 545.081,Z 130.584,A -85,B 0,C 180,E1 -3614.944,E2 -3614.944} C_VEL
LIN {X 0,Y 545.052,Z 130.587,A -85,B 0,C 180,E1 -3618.027,E2 -3618.027} C_VEL
LIN {X 0,Y 545.04,Z 130.587,A -85,B 0,C 180,E1 -3620.375,E2 -3620.375} C_VEL
LIN {X 0,Y 544.999,Z 130.595,A -85,B 0,C 180,E1 -3622.76,E2 -3622.76} C_VEL
LIN {X 0,Y 545.038,Z 130.592,A -85,B 0,C 180,E1 -3625.495,E2 -3625.495} C_VEL
LIN {X 0,Y 545.038,Z 130.589,A -85,B 0,C 180,E1 -3628.496,E2 -3628.496} C_VEL
LIN {X 0,Y 545.049,Z 130.587,A -85,B 0,C 180,E1 -3631.676,E2 -3631.676} C_VEL
LIN {X 0,Y 545.051,Z 130.589,A -85,B 0,C 180,E1 -3634.566,E2 -3634.566} C_VEL
LIN {X 0,Y 545.034,Z 130.591,A -85,B 0,C 180,E1 -3637.305,E2 -3637.305} C_VEL
LIN {X 0,Y 545.066,Z 130.585,A -85,B 0,C 180,E1 -3640.143,E2 -3640.143} C_VEL
LIN {X 0,Y 545.022,Z 130.593,A -85,B 0,C 180,E1 -3643.113,E2 -3643.113} C_VEL
LIN {X 0,Y 545.032,Z 130.591,A -85,B 0,C 180,E1 -3646.229,E2 -3646.229} C_VEL
LIN {X 0,Y 545.031,Z 130.593,A -85,B 0,C 180,E1 -3648.88,E2 -3648.88} C_VEL
LIN {X 0,Y 545.048,Z 130.587,A -85,B 0,C 180,E1 -3651.762,E2 -3651.762} C_VEL
LIN {X 0,Y 545.028,Z 130.597,A -85,B 0,C 180,E1 -3654.53,E2 -3654.53} C_VEL
LIN {X 0,Y 545.065,Z 130.584,A -85,B 0,C 180,E1 -3657.211,E2 -3657.211} C_VEL
LIN {X 0,Y 545.066,Z 130.587,A -85,B 0,C 180,E1 -3659.81,E2 -3659.81} C_VEL
LIN {X 0,Y 545.04,Z 130.592,A -85,B 0,C 180,E1 -3662.839,E2 -3662.839} C_VEL
LIN {X 0,Y 545.078,Z 130.727,A -85,B 0,C 180,E1 -3665.969,E2 -3665.969} C_VEL
LIN {X 0,Y 546.174,Z 137.764,A -85,B 0,C 180,E1 -3667.092,E2 -3667.092} C_VEL
LIN {X 0,Y 545.956,Z 154.846,A -85,B 0,C 180,E1 -3669.661,E2 -3669.661} C_VEL
LIN {X 0,Y 545.573,Z 174.259,A -85,B 0,C 180,E1 -3672.532,E2 -3672.532} C_VEL
LIN {X 0,Y 545.322,Z 192.123,A -85,B 0,C 180,E1 -3675.148,E2 -3675.148} C_VEL
LIN {X 0,Y 545.331,Z 194.12,A -85,B 0,C 180,E1 -3675.44,E2 -3675.44} C_VEL
LIN {X 0,Y 546.472,Z 203.428,A -85,B 0,C 180,E1 -3675.596,E2 -3675.596} C_VEL
LIN {X 0,Y 546.219,Z 302.308,A -85,B 0,C 180,E1 -3676.916,E2 -3676.916} C_VEL
LIN {X 0,Y 546.038,Z 315.645,A -85,B 0,C 180,E1 -3677.243,E2 -3677.243} C_VEL
LIN {X 0,Y 545.859,Z 327.848,A -85,B 0,C 180,E1 -3677.687,E2 -3677.687} C_VEL
LIN {X 0,Y 545.681,Z 339.196,A -85,B 0,C 180,E1 -3678.241,E2 -3678.241} C_VEL
LIN {X 0,Y 545.504,Z 350.49,A -85,B 0,C 180,E1 -3678.951,E2 -3678.951} C_VEL
LIN {X 0,Y 545.248,Z 361.177,A -85,B 0,C 180,E1 -3679.791,E2 -3679.791} C_VEL
LIN {X 0,Y 545.088,Z 370.81,A -85,B 0,C 180,E1 -3680.725,E2 -3680.725} C_VEL
LIN {X 0,Y 544.947,Z 378.707,A -85,B 0,C 180,E1 -3681.657,E2 -3681.657} C_VEL
LIN {X 0,Y 544.824,Z 386.419,A -85,B 0,C 180,E1 -3682.775,E2 -3682.775} C_VEL
LIN {X 0,Y 544.777,Z 393.53,A -85,B 0,C 180,E1 -3684.076,E2 -3684.076} C_VEL
LIN {X 0,Y 544.629,Z 398.255,A -85,B 0,C 180,E1 -3685.188,E2 -3685.188} C_VEL
LIN {X 0,Y 544.669,Z 401.871,A -85,B 0,C 180,E1 -3686.301,E2 -3686.301} C_VEL
LIN {X 0,Y 544.65,Z 403.734,A -85,B 0,C 180,E1 -3687.041,E2 -3687.041} C_VEL
LIN {X 0,Y 544.546,Z 406.126,A -85,B 0,C 180,E1 -3688.521,E2 -3688.521} C_VEL
LIN {X 0,Y 544.542,Z 406.735,A -85,B 0,C 180,E1 -3689.26,E2 -3689.26} C_VEL
LIN {X 0,Y 544.541,Z 406.951,A -85,B 0,C 180,E1 -3690,E2 -3690} C_VEL
LIN {X 0,Y 544.542,Z 406.735,A -85,B 0,C 180,E1 -3690.739,E2 -3690.739} C_VEL
LIN {X 0,Y 544.572,Z 405.132,A -85,B 0,C 180,E1 -3692.219,E2 -3692.219} C_VEL
LIN {X 0,Y 544.65,Z 403.738,A -85,B 0,C 180,E1 -3692.959,E2 -3692.959} C_VEL
LIN {X 0,Y 544.684,Z 400.8,A -85,B 0,C 180,E1 -3694.069,E2 -3694.069} C_VEL
LIN {X 0,Y 544.653,Z 396.818,A -85,B 0,C 180,E1 -3695.182,E2 -3695.182} C_VEL
LIN {X 0,Y 544.711,Z 391.535,A -85,B 0,C 180,E1 -3696.328,E2 -3696.328} C_VEL
LIN {X 0,Y 544.837,Z 385.251,A -85,B 0,C 180,E1 -3697.411,E2 -3697.411} C_VEL
LIN {X 0,Y 544.988,Z 377.208,A -85,B 0,C 180,E1 -3698.528,E2 -3698.528} C_VEL
LIN {X 0,Y 545.114,Z 369.01,A -85,B 0,C 180,E1 -3699.461,E2 -3699.461} C_VEL
LIN {X 0,Y 545.35,Z 359.016,A -85,B 0,C 180,E1 -3700.394,E2 -3700.394} C_VEL
LIN {X 0,Y 545.548,Z 348.151,A -85,B 0,C 180,E1 -3701.208,E2 -3701.208} C_VEL
LIN {X 0,Y 545.71,Z 336.672,A -85,B 0,C 180,E1 -3701.891,E2 -3701.891} C_VEL
LIN {X 0,Y 545.93,Z 324.42,A -85,B 0,C 180,E1 -3702.452,E2 -3702.452} C_VEL
LIN {X 0,Y 546.107,Z 311.551,A -85,B 0,C 180,E1 -3702.873,E2 -3702.873} C_VEL
LIN {X 0,Y 546.272,Z 297.893,A -85,B 0,C 180,E1 -3703.153,E2 -3703.153} C_VEL
LIN {X 0,Y 546.335,Z 200.779,A -85,B 0,C 180,E1 -3704.443,E2 -3704.443} C_VEL
LIN {X 0,Y 545.317,Z 193.923,A -85,B 0,C 180,E1 -3704.579,E2 -3704.579} C_VEL
LIN {X 0,Y 545.545,Z 174.188,A -85,B 0,C 180,E1 -3707.459,E2 -3707.459} C_VEL
LIN {X 0,Y 545.917,Z 154.649,A -85,B 0,C 180,E1 -3710.34,E2 -3710.34} C_VEL
LIN {X 0,Y 546.157,Z 137.487,A -85,B 0,C 180,E1 -3712.908,E2 -3712.908} C_VEL
LIN {X 0,Y 545.058,Z 130.594,A -85,B 0,C 180,E1 -3714.024,E2 -3714.024} C_VEL
LIN {X 0,Y 545.037,Z 130.593,A -85,B 0,C 180,E1 -3717.161,E2 -3717.161} C_VEL
LIN {X 0,Y 545.064,Z 130.588,A -85,B 0,C 180,E1 -3720.19,E2 -3720.19} C_VEL
LIN {X 0,Y 545.073,Z 130.587,A -85,B 0,C 180,E1 -3723.061,E2 -3723.061} C_VEL
LIN {X 0,Y 545.022,Z 130.596,A -85,B 0,C 180,E1 -3725.671,E2 -3725.671} C_VEL
LIN {X 0,Y 545.046,Z 130.588,A -85,B 0,C 180,E1 -3728.238,E2 -3728.238} C_VEL
LIN {X 0,Y 545.013,Z 130.597,A -85,B 0,C 180,E1 -3731.121,E2 -3731.121} C_VEL
LIN {X 0,Y 545.033,Z 130.588,A -85,B 0,C 180,E1 -3734.132,E2 -3734.132} C_VEL
LIN {X 0,Y 545.018,Z 130.597,A -85,B 0,C 180,E1 -3736.887,E2 -3736.887} C_VEL
LIN {X 0,Y 545.031,Z 130.589,A -85,B 0,C 180,E1 -3739.854,E2 -3739.854} C_VEL
LIN {X 0,Y 545.004,Z 130.598,A -85,B 0,C 180,E1 -3742.693,E2 -3742.693} C_VEL
LIN {X 0,Y 545.039,Z 130.586,A -85,B 0,C 180,E1 -3745.614,E2 -3745.614} C_VEL
LIN {X 0,Y 545.045,Z 130.591,A -85,B 0,C 180,E1 -3748.324,E2 -3748.324} C_VEL
LIN {X 0,Y 545.033,Z 130.588,A -85,B 0,C 180,E1 -3751.503,E2 -3751.503} C_VEL
LIN {X 0,Y 545.024,Z 130.598,A -85,B 0,C 180,E1 -3754.508,E2 -3754.508} C_VEL
LIN {X 0,Y 544.989,Z 130.591,A -85,B 0,C 180,E1 -3757.24,E2 -3757.24} C_VEL
LIN {X 0,Y 545.006,Z 130.593,A -85,B 0,C 180,E1 -3759.624,E2 -3759.624} C_VEL
LIN {X 0,Y 545.033,Z 130.59,A -85,B 0,C 180,E1 -3762.748,E2 -3762.748} C_VEL
LIN {X 0,Y 545.068,Z 130.589,A -85,B 0,C 180,E1 -3765.819,E2 -3765.819} C_VEL
LIN {X 0,Y 545.077,Z 130.583,A -85,B 0,C 180,E1 -3768.848,E2 -3768.848} C_VEL
LIN {X 0,Y 545.072,Z 130.59,A -85,B 0,C 180,E1 -3771.846,E2 -3771.846} C_VEL
LIN {X 0,Y 545.17,Z 130.571,A -85,B 0,C 180,E1 -3774.822,E2 -3774.822} C_VEL
LIN {X 0,Y 545.195,Z 130.576,A -85,B 0,C 180,E1 -3777.783,E2 -3777.783} C_VEL
LIN {X 0,Y 545.197,Z 130.571,A -85,B 0,C 180,E1 -3780,E2 -3780} C_VEL
LIN {X 0,Y 545.161,Z 130.573,A -85,B 0,C 180,E1 -3782.955,E2 -3782.955} C_VEL
LIN {X 0,Y 545.14,Z 130.576,A -85,B 0,C 180,E1 -3785.919,E2 -3785.919} C_VEL
LIN {X 0,Y 545.1,Z 130.583,A -85,B 0,C 180,E1 -3788.9,E2 -3788.9} C_VEL
LIN {X 0,Y 545.106,Z 130.581,A -85,B 0,C 180,E1 -3791.904,E2 -3791.904} C_VEL
LIN {X 0,Y 545.084,Z 130.587,A -85,B 0,C 180,E1 -3794.943,E2 -3794.943} C_VEL
LIN {X 0,Y 545.06,Z 130.584,A -85,B 0,C 180,E1 -3798.026,E2 -3798.026} C_VEL
LIN {X 0,Y 545.093,Z 130.583,A -85,B 0,C 180,E1 -3800.372,E2 -3800.372} C_VEL
LIN {X 0,Y 545.074,Z 130.585,A -85,B 0,C 180,E1 -3803.559,E2 -3803.559} C_VEL
LIN {X 0,Y 545.071,Z 130.584,A -85,B 0,C 180,E1 -3806,E2 -3806} C_VEL
LIN {X 0,Y 545.089,Z 130.591,A -85,B 0,C 180,E1 -3808.747,E2 -3808.747} C_VEL
LIN {X 0,Y 545.055,Z 130.587,A -85,B 0,C 180,E1 -3811.914,E2 -3811.914} C_VEL
LIN {X 0,Y 545.059,Z 130.594,A -85,B 0,C 180,E1 -3814.564,E2 -3814.564} C_VEL
LIN {X 0,Y 545.064,Z 130.588,A -85,B 0,C 180,E1 -3816.971,E2 -3816.971} C_VEL
LIN {X 0,Y 544.355,Z 130.675,A -85,B 0,C 180,E1 -3817.587,E2 -3817.587} C_VEL
LIN {X 0,Y 541.49,Z 131.036,A -85,B 0,C 180,E1 -3818.588,E2 -3818.588} C_VEL
LIN {X 0,Y 539.103,Z 131.331,A -85,B 0,C 180,E1 -3819.394,E2 -3819.394} C_VEL
LIN {X 0,Y 538.092,Z 131.458,A -85,B 0,C 180,E1 -3820.016,E2 -3820.016} C_VEL
LIN {X 0,Y 538.015,Z 131.465,A -85,B 0,C 180,E1 -3820.226,E2 -3820.226} C_VEL
LIN {X 0,Y 538.025,Z 131.465,A -85,B 0,C 180,E1 -3822.987,E2 -3822.987} C_VEL
LIN {X 0,Y 538.023,Z 131.469,A -85,B 0,C 180,E1 -3825.925,E2 -3825.925} C_VEL
LIN {X 0,Y 538.077,Z 131.459,A -85,B 0,C 180,E1 -3829.249,E2 -3829.249} C_VEL
LIN {X 0,Y 538.096,Z 131.596,A -85,B 0,C 180,E1 -3830.541,E2 -3830.541} C_VEL
LIN {X 0,Y 538.49,Z 136.902,A -85,B 0,C 180,E1 -3831.543,E2 -3831.543} C_VEL
LIN {X 0,Y 538.286,Z 154.036,A -85,B 0,C 180,E1 -3834.713,E2 -3834.713} C_VEL
LIN {X 0,Y 538.195,Z 157.197,A -85,B 0,C 180,E1 -3835.298,E2 -3835.298} C_VEL
LIN {X 0,Y 539.726,Z 166.825,A -85,B 0,C 180,E1 -3835.481,E2 -3835.481} C_VEL
LIN {X 0,Y 539.302,Z 264.165,A -85,B 0,C 180,E1 -3836.802,E2 -3836.802} C_VEL
LIN {X 0,Y 539.157,Z 277.063,A -85,B 0,C 180,E1 -3837.126,E2 -3837.126} C_VEL
LIN {X 0,Y 538.951,Z 290.346,A -85,B 0,C 180,E1 -3837.625,E2 -3837.625} C_VEL
LIN {X 0,Y 538.705,Z 302.819,A -85,B 0,C 180,E1 -3838.275,E2 -3838.275} C_VEL
LIN {X 0,Y 538.466,Z 314.667,A -85,B 0,C 180,E1 -3839.075,E2 -3839.075} C_VEL
LIN {X 0,Y 538.28,Z 324.729,A -85,B 0,C 180,E1 -3839.931,E2 -3839.931} C_VEL
LIN {X 0,Y 538.05,Z 334.033,A -85,B 0,C 180,E1 -3840.907,E2 -3840.907} C_VEL
LIN {X 0,Y 537.893,Z 342.091,A -85,B 0,C 180,E1 -3841.942,E2 -3841.942} C_VEL
LIN {X 0,Y 537.745,Z 348.762,A -85,B 0,C 180,E1 -3842.989,E2 -3842.989} C_VEL
LIN {X 0,Y 537.669,Z 354.164,A -85,B 0,C 180,E1 -3844.031,E2 -3844.031} C_VEL
LIN {X 0,Y 537.574,Z 359.253,A -85,B 0,C 180,E1 -3845.269,E2 -3845.269} C_VEL
LIN {X 0,Y 537.542,Z 362.265,A -85,B 0,C 180,E1 -3846.233,E2 -3846.233} C_VEL
LIN {X 0,Y 537.509,Z 363.953,A -85,B 0,C 180,E1 -3846.905,E2 -3846.905} C_VEL
LIN {X 0,Y 537.478,Z 366.229,A -85,B 0,C 180,E1 -3848.184,E2 -3848.184} C_VEL
LIN {X 0,Y 537.48,Z 367.251,A -85,B 0,C 180,E1 -3849.326,E2 -3849.326} C_VEL
LIN {X 0,Y 537.486,Z 367.397,A -85,B 0,C 180,E1 -3850.295,E2 -3850.295} C_VEL
LIN {X 0,Y 537.447,Z 366.455,A -85,B 0,C 180,E1 -3851.709,E2 -3851.709} C_VEL
LIN {X 0,Y 537.501,Z 365.035,A -85,B 0,C 180,E1 -3852.648,E2 -3852.648} C_VEL
LIN {X 0,Y 537.556,Z 361.669,A -85,B 0,C 180,E1 -3854.065,E2 -3854.065} C_VEL
LIN {X 0,Y 537.658,Z 357.423,A -85,B 0,C 180,E1 -3855.303,E2 -3855.303} C_VEL
LIN {X 0,Y 537.714,Z 351.558,A -85,B 0,C 180,E1 -3856.585,E2 -3856.585} C_VEL
LIN {X 0,Y 537.824,Z 344.828,A -85,B 0,C 180,E1 -3857.74,E2 -3857.74} C_VEL
LIN {X 0,Y 537.993,Z 336.483,A -85,B 0,C 180,E1 -3858.891,E2 -3858.891} C_VEL
LIN {X 0,Y 538.172,Z 327.922,A -85,B 0,C 180,E1 -3859.846,E2 -3859.846} C_VEL
LIN {X 0,Y 538.425,Z 317.349,A -85,B 0,C 180,E1 -3860.799,E2 -3860.799} C_VEL
LIN {X 0,Y 538.682,Z 306.871,A -85,B 0,C 180,E1 -3861.56,E2 -3861.56} C_VEL
LIN {X 0,Y 538.88,Z 296.457,A -85,B 0,C 180,E1 -3862.167,E2 -3862.167} C_VEL
LIN {X 0,Y 539.022,Z 283.837,A -85,B 0,C 180,E1 -3862.731,E2 -3862.731} C_VEL
LIN {X 0,Y 539.204,Z 270.308,A -85,B 0,C 180,E1 -3863.153,E2 -3863.153} C_VEL
LIN {X 0,Y 539.309,Z 256.861,A -85,B 0,C 180,E1 -3863.406,E2 -3863.406} C_VEL
LIN {X 0,Y 539.565,Z 164.789,A -85,B 0,C 180,E1 -3864.64,E2 -3864.64} C_VEL
LIN {X 0,Y 538.226,Z 157.1,A -85,B 0,C 180,E1 -3864.803,E2 -3864.803} C_VEL
LIN {X 0,Y 538.434,Z 141.353,A -85,B 0,C 180,E1 -3867.756,E2 -3867.756} C_VEL
LIN {X 0,Y 538.328,Z 133.433,A -85,B 0,C 180,E1 -3869.252,E2 -3869.252} C_VEL
LIN {X 0,Y 538.105,Z 131.46,A -85,B 0,C 180,E1 -3869.673,E2 -3869.673} C_VEL
LIN {X 0,Y 538.157,Z 131.453,A -85,B 0,C 180,E1 -3872.245,E2 -3872.245} C_VEL
LIN {X 0,Y 538.115,Z 131.451,A -85,B 0,C 180,E1 -3875.246,E2 -3875.246} C_VEL
LIN {X 0,Y 538.029,Z 131.464,A -85,B 0,C 180,E1 -3878.261,E2 -3878.261} C_VEL
LIN {X 0,Y 538.034,Z 131.466,A -85,B 0,C 180,E1 -3881.574,E2 -3881.574} C_VEL
LIN {X 0,Y 538.016,Z 131.462,A -85,B 0,C 180,E1 -3884.841,E2 -3884.841} C_VEL
LIN {X 0,Y 538.009,Z 131.471,A -85,B 0,C 180,E1 -3887.524,E2 -3887.524} C_VEL
LIN {X 0,Y 537.967,Z 131.468,A -85,B 0,C 180,E1 -3890.655,E2 -3890.655} C_VEL
LIN {X 0,Y 537.97,Z 131.471,A -85,B 0,C 180,E1 -3893.074,E2 -3893.074} C_VEL
LIN {X 0,Y 537.973,Z 131.473,A -85,B 0,C 180,E1 -3895.658,E2 -3895.658} C_VEL
LIN {X 0,Y 537.966,Z 131.469,A -85,B 0,C 180,E1 -3898.054,E2 -3898.054} C_VEL
LIN {X 0,Y 537.984,Z 131.467,A -85,B 0,C 180,E1 -3900.63,E2 -3900.63} C_VEL
LIN {X 0,Y 537.996,Z 131.474,A -85,B 0,C 180,E1 -3903.275,E2 -3903.275} C_VEL
LIN {X 0,Y 537.949,Z 131.471,A -85,B 0,C 180,E1 -3906.009,E2 -3906.009} C_VEL
LIN {X 0,Y 537.981,Z 131.471,A -85,B 0,C 180,E1 -3908.834,E2 -3908.834} C_VEL
LIN {X 0,Y 537.974,Z 131.468,A -85,B 0,C 180,E1 -3911.873,E2 -3911.873} C_VEL
LIN {X 0,Y 537.992,Z 131.473,A -85,B 0,C 180,E1 -3914.864,E2 -3914.864} C_VEL
LIN {X 0,Y 537.968,Z 131.473,A -85,B 0,C 180,E1 -3917.21,E2 -3917.21} C_VEL
LIN {X 0,Y 537.986,Z 131.467,A -85,B 0,C 180,E1 -3920.2,E2 -3920.2} C_VEL
LIN {X 0,Y 537.972,Z 131.472,A -85,B 0,C 180,E1 -3923.063,E2 -3923.063} C_VEL
LIN {X 0,Y 537.988,Z 131.466,A -85,B 0,C 180,E1 -3925.825,E2 -3925.825} C_VEL
LIN {X 0,Y 537.99,Z 131.473,A -85,B 0,C 180,E1 -3928.498,E2 -3928.498} C_VEL
LIN {X 0,Y 537.986,Z 131.468,A -85,B 0,C 180,E1 -3931.096,E2 -3931.096} C_VEL
LIN {X 0,Y 537.981,Z 131.467,A -85,B 0,C 180,E1 -3933.631,E2 -3933.631} C_VEL
LIN {X 0,Y 537.985,Z 131.471,A -85,B 0,C 180,E1 -3936.129,E2 -3936.129} C_VEL
LIN {X 0,Y 537.99,Z 131.472,A -85,B 0,C 180,E1 -3938.545,E2 -3938.545} C_VEL
LIN {X 0,Y 537.959,Z 131.471,A -85,B 0,C 180,E1 -3940.938,E2 -3940.938} C_VEL
LIN {X 0,Y 537.97,Z 131.468,A -85,B 0,C 180,E1 -3943.298,E2 -3943.298} C_VEL
LIN {X 0,Y 538.033,Z 131.462,A -85,B 0,C 180,E1 -3945.63,E2 -3945.63} C_VEL
LIN {X 0,Y 538.027,Z 131.462,A -85,B 0,C 180,E1 -3948.701,E2 -3948.701} C_VEL
LIN {X 0,Y 538.038,Z 131.464,A -85,B 0,C 180,E1 -3951.739,E2 -3951.739} C_VEL
LIN {X 0,Y 538.123,Z 131.449,A -85,B 0,C 180,E1 -3954.755,E2 -3954.755} C_VEL
LIN {X 0,Y 538.165,Z 131.451,A -85,B 0,C 180,E1 -3957.755,E2 -3957.755} C_VEL
LIN {X 0,Y 538.163,Z 131.451,A -85,B 0,C 180,E1 -3960,E2 -3960} C_VEL
LIN {X 0,Y 538.113,Z 131.451,A -85,B 0,C 180,E1 -3962.995,E2 -3962.995} C_VEL
LIN {X 0,Y 538.079,Z 131.459,A -85,B 0,C 180,E1 -3965.998,E2 -3965.998} C_VEL
LIN {X 0,Y 538.031,Z 131.462,A -85,B 0,C 180,E1 -3969.019,E2 -3969.019} C_VEL
LIN {X 0,Y 538.055,Z 131.459,A -85,B 0,C 180,E1 -3972.064,E2 -3972.064} C_VEL
LIN {X 0,Y 538.041,Z 131.464,A -85,B 0,C 180,E1 -3975.144,E2 -3975.144} C_VEL
LIN {X 0,Y 538.007,Z 131.463,A -85,B 0,C 180,E1 -3978.271,E2 -3978.271} C_VEL
LIN {X 0,Y 537.997,Z 131.466,A -85,B 0,C 180,E1 -3980.653,E2 -3980.653} C_VEL
LIN {X 0,Y 537.984,Z 131.473,A -85,B 0,C 180,E1 -3983.074,E2 -3983.074} C_VEL
LIN {X 0,Y 537.997,Z 131.467,A -85,B 0,C 180,E1 -3985.661,E2 -3985.661} C_VEL
LIN {X 0,Y 537.977,Z 131.467,A -85,B 0,C 180,E1 -3988.054,E2 -3988.054} C_VEL
LIN {X 0,Y 537.993,Z 131.468,A -85,B 0,C 180,E1 -3990.629,E2 -3990.629} C_VEL
LIN {X 0,Y 538.025,Z 131.466,A -85,B 0,C 180,E1 -3993.278,E2 -3993.278} C_VEL
LIN {X 0,Y 537.993,Z 131.465,A -85,B 0,C 180,E1 -3996.005,E2 -3996.005} C_VEL
LIN {X 0,Y 538.013,Z 131.472,A -85,B 0,C 180,E1 -3998.831,E2 -3998.831} C_VEL
LIN {X 0,Y 537.992,Z 131.465,A -85,B 0,C 180,E1 -4001.873,E2 -4001.873} C_VEL
LIN {X 0,Y 537.998,Z 131.471,A -85,B 0,C 180,E1 -4004.864,E2 -4004.864} C_VEL
LIN {X 0,Y 537.977,Z 131.469,A -85,B 0,C 180,E1 -4007.209,E2 -4007.209} C_VEL
LIN {X 0,Y 538.011,Z 131.466,A -85,B 0,C 180,E1 -4010.201,E2 -4010.201} C_VEL
LIN {X 0,Y 538.021,Z 131.463,A -85,B 0,C 180,E1 -4013.066,E2 -4013.066} C_VEL
LIN {X 0,Y 538.001,Z 131.465,A -85,B 0,C 180,E1 -4015.825,E2 -4015.825} C_VEL
LIN {X 0,Y 538.012,Z 131.471,A -85,B 0,C 180,E1 -4018.498,E2 -4018.498} C_VEL
LIN {X 0,Y 538.005,Z 131.465,A -85,B 0,C 180,E1 -4021.096,E2 -4021.096} C_VEL
LIN {X 0,Y 537.993,Z 131.47,A -85,B 0,C 180,E1 -4023.63,E2 -4023.63} C_VEL
LIN {X 0,Y 538.046,Z 131.654,A -85,B 0,C 180,E1 -4025.816,E2 -4025.816} C_VEL
LIN {X 0,Y 539.233,Z 138.85,A -85,B 0,C 180,E1 -4026.983,E2 -4026.983} C_VEL
LIN {X 0,Y 538.938,Z 156.653,A -85,B 0,C 180,E1 -4029.696,E2 -4029.696} C_VEL
LIN {X 0,Y 538.565,Z 175.598,A -85,B 0,C 180,E1 -4032.534,E2 -4032.534} C_VEL
LIN {X 0,Y 538.268,Z 193.803,A -85,B 0,C 180,E1 -4035.235,E2 -4035.235} C_VEL
LIN {X 0,Y 539.6,Z 203.616,A -85,B 0,C 180,E1 -4035.415,E2 -4035.415} C_VEL
LIN {X 0,Y 539.323,Z 301.993,A -85,B 0,C 180,E1 -4036.746,E2 -4036.746} C_VEL
LIN {X 0,Y 539.113,Z 315.351,A -85,B 0,C 180,E1 -4037.076,E2 -4037.076} C_VEL
LIN {X 0,Y 538.905,Z 327.563,A -85,B 0,C 180,E1 -4037.526,E2 -4037.526} C_VEL
LIN {X 0,Y 538.689,Z 339.476,A -85,B 0,C 180,E1 -4038.118,E2 -4038.118} C_VEL
LIN {X 0,Y 538.479,Z 351.514,A -85,B 0,C 180,E1 -4038.9,E2 -4038.9} C_VEL
LIN {X 0,Y 538.198,Z 361.981,A -85,B 0,C 180,E1 -4039.751,E2 -4039.751} C_VEL
LIN {X 0,Y 538.048,Z 370.543,A -85,B 0,C 180,E1 -4040.603,E2 -4040.603} C_VEL
LIN {X 0,Y 537.9,Z 378.442,A -85,B 0,C 180,E1 -4041.547,E2 -4041.547} C_VEL
LIN {X 0,Y 537.755,Z 386.157,A -85,B 0,C 180,E1 -4042.679,E2 -4042.679} C_VEL
LIN {X 0,Y 537.666,Z 393.268,A -85,B 0,C 180,E1 -4043.997,E2 -4043.997} C_VEL
LIN {X 0,Y 537.54,Z 397.996,A -85,B 0,C 180,E1 -4045.125,E2 -4045.125} C_VEL
LIN {X 0,Y 537.591,Z 401.613,A -85,B 0,C 180,E1 -4046.252,E2 -4046.252} C_VEL
LIN {X 0,Y 537.551,Z 403.476,A -85,B 0,C 180,E1 -4047.002,E2 -4047.002} C_VEL
LIN {X 0,Y 537.451,Z 405.867,A -85,B 0,C 180,E1 -4048.501,E2 -4048.501} C_VEL
LIN {X 0,Y 537.446,Z 406.476,A -85,B 0,C 180,E1 -4049.251,E2 -4049.251} C_VEL
LIN {X 0,Y 537.447,Z 406.692,A -85,B 0,C 180,E1 -4050,E2 -4050} C_VEL
LIN {X 0,Y 537.446,Z 406.476,A -85,B 0,C 180,E1 -4050.749,E2 -4050.749} C_VEL
LIN {X 0,Y 537.49,Z 404.872,A -85,B 0,C 180,E1 -4052.248,E2 -4052.248} C_VEL
LIN {X 0,Y 537.551,Z 403.475,A -85,B 0,C 180,E1 -4052.998,E2 -4052.998} C_VEL
LIN {X 0,Y 537.603,Z 400.536,A -85,B 0,C 180,E1 -4054.123,E2 -4054.123} C_VEL
LIN {X 0,Y 537.587,Z 396.553,A -85,B 0,C 180,E1 -4055.251,E2 -4055.251} C_VEL
LIN {X 0,Y 537.645,Z 390.497,A -85,B 0,C 180,E1 -4056.555,E2 -4056.555} C_VEL
LIN {X 0,Y 537.784,Z 383.739,A -85,B 0,C 180,E1 -4057.698,E2 -4057.698} C_VEL
LIN {X 0,Y 537.933,Z 375.436,A -85,B 0,C 180,E1 -4058.83,E2 -4058.83} C_VEL
LIN {X 0,Y 538.101,Z 366.925,A -85,B 0,C 180,E1 -4059.776,E2 -4059.776} C_VEL
LIN {X 0,Y 538.36,Z 356.412,A -85,B 0,C 180,E1 -4060.721,E2 -4060.721} C_VEL
LIN {X 0,Y 538.582,Z 345.211,A -85,B 0,C 180,E1 -4061.532,E2 -4061.532} C_VEL
LIN {X 0,Y 538.813,Z 334.606,A -85,B 0,C 180,E1 -4062.141,E2 -4062.141} C_VEL
LIN {X 0,Y 538.985,Z 322.892,A -85,B 0,C 180,E1 -4062.663,E2 -4062.663} C_VEL
LIN {X 0,Y 539.173,Z 309.397,A -85,B 0,C 180,E1 -4063.09,E2 -4063.09} C_VEL
LIN {X 0,Y 539.368,Z 295.996,A -85,B 0,C 180,E1 -4063.349,E2 -4063.349} C_VEL
LIN {X 0,Y 539.459,Z 201.544,A -85,B 0,C 180,E1 -4064.617,E2 -4064.617} C_VEL
LIN {X 0,Y 538.236,Z 193.61,A -85,B 0,C 180,E1 -4064.781,E2 -4064.781} C_VEL
LIN {X 0,Y 538.54,Z 175.43,A -85,B 0,C 180,E1 -4067.467,E2 -4067.467} C_VEL
LIN {X 0,Y 538.94,Z 155.405,A -85,B 0,C 180,E1 -4070.458,E2 -4070.458} C_VEL
LIN {X 0,Y 539.201,Z 138.529,A -85,B 0,C 180,E1 -4073.018,E2 -4073.018} C_VEL
LIN {X 0,Y 538.021,Z 131.47,A -85,B 0,C 180,E1 -4074.184,E2 -4074.184} C_VEL
LIN {X 0,Y 538.01,Z 131.469,A -85,B 0,C 180,E1 -4077.207,E2 -4077.207} C_VEL
LIN {X 0,Y 538.001,Z 131.473,A -85,B 0,C 180,E1 -4079.762,E2 -4079.762} C_VEL
LIN {X 0,Y 538.016,Z 131.464,A -85,B 0,C 180,E1 -4082.383,E2 -4082.383} C_VEL
LIN {X 0,Y 537.988,Z 131.469,A -85,B 0,C 180,E1 -4085.085,E2 -4085.085} C_VEL
LIN {X 0,Y 537.986,Z 131.469,A -85,B 0,C 180,E1 -4087.878,E2 -4087.878} C_VEL
LIN {X 0,Y 537.994,Z 131.468,A -85,B 0,C 180,E1 -4090.781,E2 -4090.781} C_VEL
LIN {X 0,Y 538.003,Z 131.464,A -85,B 0,C 180,E1 -4094.071,E2 -4094.071} C_VEL
LIN {X 0,Y 537.971,Z 131.476,A -85,B 0,C 180,E1 -4097.019,E2 -4097.019} C_VEL
LIN {X 0,Y 537.991,Z 131.471,A -85,B 0,C 180,E1 -4099.26,E2 -4099.26} C_VEL
LIN {X 0,Y 537.966,Z 131.469,A -85,B 0,C 180,E1 -4102.12,E2 -4102.12} C_VEL
LIN {X 0,Y 537.985,Z 131.466,A -85,B 0,C 180,E1 -4105.387,E2 -4105.387} C_VEL
LIN {X 0,Y 537.995,Z 131.467,A -85,B 0,C 180,E1 -4108.116,E2 -4108.116} C_VEL
LIN {X 0,Y 537.987,Z 131.468,A -85,B 0,C 180,E1 -4111.095,E2 -4111.095} C_VEL
LIN {X 0,Y 537.979,Z 131.465,A -85,B 0,C 180,E1 -4113.63,E2 -4113.63} C_VEL
LIN {X 0,Y 537.986,Z 131.471,A -85,B 0,C 180,E1 -4116.128,E2 -4116.128} C_VEL
LIN {X 0,Y 537.991,Z 131.472,A -85,B 0,C 180,E1 -4118.544,E2 -4118.544} C_VEL
LIN {X 0,Y 537.96,Z 131.469,A -85,B 0,C 180,E1 -4120.937,E2 -4120.937} C_VEL
LIN {X 0,Y 537.972,Z 131.467,A -85,B 0,C 180,E1 -4123.297,E2 -4123.297} C_VEL
LIN {X 0,Y 538.041,Z 131.462,A -85,B 0,C 180,E1 -4125.63,E2 -4125.63} C_VEL
LIN {X 0,Y 538.028,Z 131.462,A -85,B 0,C 180,E1 -4128.7,E2 -4128.7} C_VEL
LIN {X 0,Y 538.043,Z 131.464,A -85,B 0,C 180,E1 -4131.739,E2 -4131.739} C_VEL
LIN {X 0,Y 538.129,Z 131.448,A -85,B 0,C 180,E1 -4134.754,E2 -4134.754} C_VEL
LIN {X 0,Y 538.166,Z 131.451,A -85,B 0,C 180,E1 -4137.754,E2 -4137.754} C_VEL
LIN {X 0,Y 538.166,Z 131.446,A -85,B 0,C 180,E1 -4140,E2 -4140} C_VEL
LIN {X 0,Y 538.129,Z 131.449,A -85,B 0,C 180,E1 -4142.994,E2 -4142.994} C_VEL
LIN {X 0,Y 538.095,Z 131.453,A -85,B 0,C 180,E1 -4145.997,E2 -4145.997} C_VEL
LIN {X 0,Y 538.053,Z 131.462,A -85,B 0,C 180,E1 -4149.017,E2 -4149.017} C_VEL
LIN {X 0,Y 538.065,Z 131.457,A -85,B 0,C 180,E1 -4152.062,E2 -4152.062} C_VEL
LIN {X 0,Y 538.044,Z 131.466,A -85,B 0,C 180,E1 -4155.143,E2 -4155.143} C_VEL
LIN {X 0,Y 538.013,Z 131.462,A -85,B 0,C 180,E1 -4158.27,E2 -4158.27} C_VEL
LIN {X 0,Y 538.038,Z 131.465,A -85,B 0,C 180,E1 -4160.651,E2 -4160.651} C_VEL
LIN {X 0,Y 538.007,Z 131.464,A -85,B 0,C 180,E1 -4163.877,E2 -4163.877} C_VEL
LIN {X 0,Y 538.037,Z 131.463,A -85,B 0,C 180,E1 -4166.366,E2 -4166.366} C_VEL
LIN {X 0,Y 538.03,Z 131.467,A -85,B 0,C 180,E1 -4168.933,E2 -4168.933} C_VEL
LIN {X 0,Y 538.01,Z 131.465,A -85,B 0,C 180,E1 -4171.887,E2 -4171.887} C_VEL
LIN {X 0,Y 538.009,Z 131.472,A -85,B 0,C 180,E1 -4174.617,E2 -4174.617} C_VEL
LIN {X 0,Y 538.004,Z 131.467,A -85,B 0,C 180,E1 -4177.169,E2 -4177.169} C_VEL
LIN {X 0,Y 538.015,Z 131.465,A -85,B 0,C 180,E1 -4180.226,E2 -4180.226} C_VEL
LIN {X 0,Y 537.366,Z 131.549,A -85,B 0,C 180,E1 -4180.852,E2 -4180.852} C_VEL
LIN {X 0,Y 534.52,Z 131.904,A -85,B 0,C 180,E1 -4181.867,E2 -4181.867} C_VEL
LIN {X 0,Y 532.099,Z 132.206,A -85,B 0,C 180,E1 -4182.684,E2 -4182.684} C_VEL
LIN {X 0,Y 531.052,Z 132.335,A -85,B 0,C 180,E1 -4183.315,E2 -4183.315} C_VEL
LIN {X 0,Y 530.962,Z 132.345,A -85,B 0,C 180,E1 -4183.528,E2 -4183.528} C_VEL
LIN {X 0,Y 530.958,Z 132.348,A -85,B 0,C 180,E1 -4186.504,E2 -4186.504} C_VEL
LIN {X 0,Y 531.004,Z 132.343,A -85,B 0,C 180,E1 -4189.569,E2 -4189.569} C_VEL
LIN {X 0,Y 531.044,Z 132.356,A -85,B 0,C 180,E1 -4190.407,E2 -4190.407} C_VEL
LIN {X 0,Y 531.502,Z 136.9,A -85,B 0,C 180,E1 -4191.274,E2 -4191.274} C_VEL
LIN {X 0,Y 531.318,Z 152.047,A -85,B 0,C 180,E1 -4194.098,E2 -4194.098} C_VEL
LIN {X 0,Y 531.221,Z 157.489,A -85,B 0,C 180,E1 -4195.109,E2 -4195.109} C_VEL
LIN {X 0,Y 532.864,Z 167.053,A -85,B 0,C 180,E1 -4195.289,E2 -4195.289} C_VEL
LIN {X 0,Y 532.416,Z 264.383,A -85,B 0,C 180,E1 -4196.628,E2 -4196.628} C_VEL
LIN {X 0,Y 532.278,Z 276.868,A -85,B 0,C 180,E1 -4196.943,E2 -4196.943} C_VEL
LIN {X 0,Y 532.037,Z 290.109,A -85,B 0,C 180,E1 -4197.44,E2 -4197.44} C_VEL
LIN {X 0,Y 531.782,Z 301.495,A -85,B 0,C 180,E1 -4198.023,E2 -4198.023} C_VEL
LIN {X 0,Y 531.597,Z 312.379,A -85,B 0,C 180,E1 -4198.741,E2 -4198.741} C_VEL
LIN {X 0,Y 531.307,Z 323.432,A -85,B 0,C 180,E1 -4199.652,E2 -4199.652} C_VEL
LIN {X 0,Y 531.1,Z 331.502,A -85,B 0,C 180,E1 -4200.467,E2 -4200.467} C_VEL
LIN {X 0,Y 530.903,Z 340.271,A -85,B 0,C 180,E1 -4201.539,E2 -4201.539} C_VEL
LIN {X 0,Y 530.717,Z 347.849,A -85,B 0,C 180,E1 -4202.693,E2 -4202.693} C_VEL
LIN {X 0,Y 530.635,Z 353.054,A -85,B 0,C 180,E1 -4203.66,E2 -4203.66} C_VEL
LIN {X 0,Y 530.498,Z 358.443,A -85,B 0,C 180,E1 -4204.917,E2 -4204.917} C_VEL
LIN {X 0,Y 530.458,Z 362.262,A -85,B 0,C 180,E1 -4206.088,E2 -4206.088} C_VEL
LIN {X 0,Y 530.402,Z 365.295,A -85,B 0,C 180,E1 -4207.402,E2 -4207.402} C_VEL
LIN {X 0,Y 530.405,Z 366.573,A -85,B 0,C 180,E1 -4208.222,E2 -4208.222} C_VEL
LIN {X 0,Y 530.373,Z 367.336,A -85,B 0,C 180,E1 -4209.036,E2 -4209.036} C_VEL
LIN {X 0,Y 530.398,Z 367.68,A -85,B 0,C 180,E1 -4210.181,E2 -4210.181} C_VEL
LIN {X 0,Y 530.364,Z 367.001,A -85,B 0,C 180,E1 -4211.456,E2 -4211.456} C_VEL
LIN {X 0,Y 530.403,Z 365.532,A -85,B 0,C 180,E1 -4212.556,E2 -4212.556} C_VEL
LIN {X 0,Y 530.44,Z 362.685,A -85,B 0,C 180,E1 -4213.845,E2 -4213.845} C_VEL
LIN {X 0,Y 530.59,Z 358.24,A -85,B 0,C 180,E1 -4215.222,E2 -4215.222} C_VEL
LIN {X 0,Y 530.639,Z 352.2,A -85,B 0,C 180,E1 -4216.598,E2 -4216.598} C_VEL
LIN {X 0,Y 530.788,Z 345.545,A -85,B 0,C 180,E1 -4217.769,E2 -4217.769} C_VEL
LIN {X 0,Y 530.972,Z 337.294,A -85,B 0,C 180,E1 -4218.935,E2 -4218.935} C_VEL
LIN {X 0,Y 531.159,Z 328.874,A -85,B 0,C 180,E1 -4219.903,E2 -4219.903} C_VEL
LIN {X 0,Y 531.414,Z 318.485,A -85,B 0,C 180,E1 -4220.869,E2 -4220.869} C_VEL
LIN {X 0,Y 531.712,Z 308.178,A -85,B 0,C 180,E1 -4221.64,E2 -4221.64} C_VEL
LIN {X 0,Y 531.95,Z 296.932,A -85,B 0,C 180,E1 -4222.314,E2 -4222.314} C_VEL
LIN {X 0,Y 532.107,Z 284.677,A -85,B 0,C 180,E1 -4222.876,E2 -4222.876} C_VEL
LIN {X 0,Y 532.278,Z 271.73,A -85,B 0,C 180,E1 -4223.294,E2 -4223.294} C_VEL
LIN {X 0,Y 532.452,Z 258.609,A -85,B 0,C 180,E1 -4223.558,E2 -4223.558} C_VEL
LIN {X 0,Y 532.723,Z 165.882,A -85,B 0,C 180,E1 -4224.82,E2 -4224.82} C_VEL
LIN {X 0,Y 531.239,Z 157.371,A -85,B 0,C 180,E1 -4224.996,E2 -4224.996} C_VEL
LIN {X 0,Y 531.438,Z 140.898,A -85,B 0,C 180,E1 -4228.106,E2 -4228.106} C_VEL
LIN {X 0,Y 531.386,Z 134.937,A -85,B 0,C 180,E1 -4229.242,E2 -4229.242} C_VEL
LIN {X 0,Y 531.093,Z 132.334,A -85,B 0,C 180,E1 -4229.763,E2 -4229.763} C_VEL
LIN {X 0,Y 531.129,Z 132.329,A -85,B 0,C 180,E1 -4232.275,E2 -4232.275} C_VEL
LIN {X 0,Y 531.076,Z 132.328,A -85,B 0,C 180,E1 -4235.315,E2 -4235.315} C_VEL
LIN {X 0,Y 530.977,Z 132.341,A -85,B 0,C 180,E1 -4238.372,E2 -4238.372} C_VEL
LIN {X 0,Y 531.006,Z 132.342,A -85,B 0,C 180,E1 -4241.65,E2 -4241.65} C_VEL
LIN {X 0,Y 530.969,Z 132.34,A -85,B 0,C 180,E1 -4244.932,E2 -4244.932} C_VEL
LIN {X 0,Y 530.965,Z 132.349,A -85,B 0,C 180,E1 -4247.724,E2 -4247.724} C_VEL
LIN {X 0,Y 530.925,Z 132.347,A -85,B 0,C 180,E1 -4250.941,E2 -4250.941} C_VEL
LIN {X 0,Y 530.917,Z 132.354,A -85,B 0,C 180,E1 -4253.399,E2 -4253.399} C_VEL
LIN {X 0,Y 530.921,Z 132.349,A -85,B 0,C 180,E1 -4255.902,E2 -4255.902} C_VEL
LIN {X 0,Y 530.926,Z 132.345,A -85,B 0,C 180,E1 -4258.46,E2 -4258.46} C_VEL
LIN {X 0,Y 530.931,Z 132.35,A -85,B 0,C 180,E1 -4261.081,E2 -4261.081} C_VEL
LIN {X 0,Y 530.928,Z 132.347,A -85,B 0,C 180,E1 -4263.777,E2 -4263.777} C_VEL
LIN {X 0,Y 530.901,Z 132.35,A -85,B 0,C 180,E1 -4266.563,E2 -4266.563} C_VEL
LIN {X 0,Y 530.941,Z 132.348,A -85,B 0,C 180,E1 -4269.448,E2 -4269.448} C_VEL
LIN {X 0,Y 530.909,Z 132.349,A -85,B 0,C 180,E1 -4272.464,E2 -4272.464} C_VEL
LIN {X 0,Y 530.962,Z 132.343,A -85,B 0,C 180,E1 -4275.451,E2 -4275.451} C_VEL
LIN {X 0,Y 530.946,Z 132.347,A -85,B 0,C 180,E1 -4278.561,E2 -4278.561} C_VEL
LIN {X 0,Y 530.945,Z 132.344,A -85,B 0,C 180,E1 -4281.529,E2 -4281.529} C_VEL
LIN {X 0,Y 530.928,Z 132.349,A -85,B 0,C 180,E1 -4284.379,E2 -4284.379} C_VEL
LIN {X 0,Y 530.945,Z 132.346,A -85,B 0,C 180,E1 -4287.132,E2 -4287.132} C_VEL
LIN {X 0,Y 530.93,Z 132.345,A -85,B 0,C 180,E1 -4289.801,E2 -4289.801} C_VEL
LIN {X 0,Y 530.956,Z 132.35,A -85,B 0,C 180,E1 -4292.481,E2 -4292.481} C_VEL
LIN {X 0,Y 530.948,Z 132.344,A -85,B 0,C 180,E1 -4295.774,E2 -4295.774} C_VEL
LIN {X 0,Y 530.949,Z 132.35,A -85,B 0,C 180,E1 -4298.246,E2 -4298.246} C_VEL
LIN {X 0,Y 530.918,Z 132.35,A -85,B 0,C 180,E1 -4300.675,E2 -4300.675} C_VEL
LIN {X 0,Y 530.933,Z 132.345,A -85,B 0,C 180,E1 -4303.07,E2 -4303.07} C_VEL
LIN {X 0,Y 530.983,Z 132.339,A -85,B 0,C 180,E1 -4305.435,E2 -4305.435} C_VEL
LIN {X 0,Y 530.99,Z 132.341,A -85,B 0,C 180,E1 -4308.549,E2 -4308.549} C_VEL
LIN {X 0,Y 530.986,Z 132.341,A -85,B 0,C 180,E1 -4311.629,E2 -4311.629} C_VEL
LIN {X 0,Y 531.084,Z 132.326,A -85,B 0,C 180,E1 -4314.685,E2 -4314.685} C_VEL
LIN {X 0,Y 531.136,Z 132.326,A -85,B 0,C 180,E1 -4317.725,E2 -4317.725} C_VEL
LIN {X 0,Y 531.132,Z 132.326,A -85,B 0,C 180,E1 -4320,E2 -4320} C_VEL
LIN {X 0,Y 531.136,Z 132.322,A -85,B 0,C 180,E1 -4322.275,E2 -4322.275} C_VEL
LIN {X 0,Y 531.085,Z 132.329,A -85,B 0,C 180,E1 -4325.315,E2 -4325.315} C_VEL
LIN {X 0,Y 530.987,Z 132.338,A -85,B 0,C 180,E1 -4328.372,E2 -4328.372} C_VEL
LIN {X 0,Y 531.055,Z 132.337,A -85,B 0,C 180,E1 -4331.67,E2 -4331.67} C_VEL
LIN {X 0,Y 531.024,Z 132.335,A -85,B 0,C 180,E1 -4334.95,E2 -4334.95} C_VEL
LIN {X 0,Y 530.977,Z 132.343,A -85,B 0,C 180,E1 -4337.724,E2 -4337.724} C_VEL
LIN {X 0,Y 531.012,Z 132.335,A -85,B 0,C 180,E1 -4340.128,E2 -4340.128} C_VEL
LIN {X 0,Y 530.924,Z 132.346,A -85,B 0,C 180,E1 -4342.575,E2 -4342.575} C_VEL
LIN {X 0,Y 530.951,Z 132.349,A -85,B 0,C 180,E1 -4345.061,E2 -4345.061} C_VEL
LIN {X 0,Y 530.956,Z 132.344,A -85,B 0,C 180,E1 -4347.599,E2 -4347.599} C_VEL
LIN {X 0,Y 530.936,Z 132.344,A -85,B 0,C 180,E1 -4350.199,E2 -4350.199} C_VEL
LIN {X 0,Y 530.969,Z 132.347,A -85,B 0,C 180,E1 -4352.867,E2 -4352.867} C_VEL
LIN {X 0,Y 530.951,Z 132.343,A -85,B 0,C 180,E1 -4355.621,E2 -4355.621} C_VEL
LIN {X 0,Y 530.966,Z 132.346,A -85,B 0,C 180,E1 -4358.653,E2 -4358.653} C_VEL
LIN {X 0,Y 530.963,Z 132.342,A -85,B 0,C 180,E1 -4361.439,E2 -4361.439} C_VEL
LIN {X 0,Y 530.968,Z 132.347,A -85,B 0,C 180,E1 -4364.549,E2 -4364.549} C_VEL
LIN {X 0,Y 530.922,Z 132.346,A -85,B 0,C 180,E1 -4367.537,E2 -4367.537} C_VEL
LIN {X 0,Y 530.972,Z 132.349,A -85,B 0,C 180,E1 -4370.555,E2 -4370.555} C_VEL
LIN {X 0,Y 530.953,Z 132.342,A -85,B 0,C 180,E1 -4373.441,E2 -4373.441} C_VEL
LIN {X 0,Y 530.965,Z 132.349,A -85,B 0,C 180,E1 -4376.501,E2 -4376.501} C_VEL
LIN {X 0,Y 530.965,Z 132.342,A -85,B 0,C 180,E1 -4379.357,E2 -4379.357} C_VEL
LIN {X 0,Y 530.966,Z 132.35,A -85,B 0,C 180,E1 -4382.478,E2 -4382.478} C_VEL
LIN {X 0,Y 530.985,Z 132.346,A -85,B 0,C 180,E1 -4385.619,E2 -4385.619} C_VEL
LIN {X 0,Y 532.276,Z 139.919,A -85,B 0,C 180,E1 -4386.87,E2 -4386.87} C_VEL
LIN {X 0,Y 531.995,Z 157.018,A -85,B 0,C 180,E1 -4389.513,E2 -4389.513} C_VEL
LIN {X 0,Y 531.559,Z 176.651,A -85,B 0,C 180,E1 -4392.495,E2 -4392.495} C_VEL
LIN {X 0,Y 531.249,Z 193.567,A -85,B 0,C 180,E1 -4395.039,E2 -4395.039} C_VEL
LIN {X 0,Y 532.751,Z 204.474,A -85,B 0,C 180,E1 -4395.238,E2 -4395.238} C_VEL
LIN {X 0,Y 532.409,Z 301.677,A -85,B 0,C 180,E1 -4396.571,E2 -4396.571} C_VEL
LIN {X 0,Y 532.227,Z 314.294,A -85,B 0,C 180,E1 -4396.882,E2 -4396.882} C_VEL
LIN {X 0,Y 531.962,Z 327.278,A -85,B 0,C 180,E1 -4397.36,E2 -4397.36} C_VEL
LIN {X 0,Y 531.722,Z 339.628,A -85,B 0,C 180,E1 -4397.986,E2 -4397.986} C_VEL
LIN {X 0,Y 531.484,Z 351.241,A -85,B 0,C 180,E1 -4398.752,E2 -4398.752} C_VEL
LIN {X 0,Y 531.211,Z 361.713,A -85,B 0,C 180,E1 -4399.615,E2 -4399.615} C_VEL
LIN {X 0,Y 531.015,Z 370.276,A -85,B 0,C 180,E1 -4400.477,E2 -4400.477} C_VEL
LIN {X 0,Y 530.848,Z 378.178,A -85,B 0,C 180,E1 -4401.434,E2 -4401.434} C_VEL
LIN {X 0,Y 530.667,Z 385.894,A -85,B 0,C 180,E1 -4402.581,E2 -4402.581} C_VEL
LIN {X 0,Y 530.562,Z 393.006,A -85,B 0,C 180,E1 -4403.917,E2 -4403.917} C_VEL
LIN {X 0,Y 530.459,Z 397.736,A -85,B 0,C 180,E1 -4405.06,E2 -4405.06} C_VEL
LIN {X 0,Y 530.516,Z 401.354,A -85,B 0,C 180,E1 -4406.202,E2 -4406.202} C_VEL
LIN {X 0,Y 530.457,Z 403.217,A -85,B 0,C 180,E1 -4406.962,E2 -4406.962} C_VEL
LIN {X 0,Y 530.412,Z 404.614,A -85,B 0,C 180,E1 -4407.722,E2 -4407.722} C_VEL
LIN {X 0,Y 530.351,Z 406.217,A -85,B 0,C 180,E1 -4409.241,E2 -4409.241} C_VEL
LIN {X 0,Y 530.352,Z 406.433,A -85,B 0,C 180,E1 -4410,E2 -4410} C_VEL
LIN {X 0,Y 530.361,Z 405.608,A -85,B 0,C 180,E1 -4411.519,E2 -4411.519} C_VEL
LIN {X 0,Y 530.411,Z 404.611,A -85,B 0,C 180,E1 -4412.278,E2 -4412.278} C_VEL
LIN {X 0,Y 530.457,Z 403.213,A -85,B 0,C 180,E1 -4413.038,E2 -4413.038} C_VEL
LIN {X 0,Y 530.521,Z 400.272,A -85,B 0,C 180,E1 -4414.178,E2 -4414.178} C_VEL
LIN {X 0,Y 530.522,Z 396.287,A -85,B 0,C 180,E1 -4415.321,E2 -4415.321} C_VEL
LIN {X 0,Y 530.546,Z 390.822,A -85,B 0,C 180,E1 -4416.531,E2 -4416.531} C_VEL
LIN {X 0,Y 530.704,Z 383.467,A -85,B 0,C 180,E1 -4417.801,E2 -4417.801} C_VEL
LIN {X 0,Y 530.886,Z 375.161,A -85,B 0,C 180,E1 -4418.949,E2 -4418.949} C_VEL
LIN {X 0,Y 531.06,Z 366.645,A -85,B 0,C 180,E1 -4419.906,E2 -4419.906} C_VEL
LIN {X 0,Y 531.348,Z 356.128,A -85,B 0,C 180,E1 -4420.864,E2 -4420.864} C_VEL
LIN {X 0,Y 531.608,Z 344.321,A -85,B 0,C 180,E1 -4421.726,E2 -4421.726} C_VEL
LIN {X 0,Y 531.868,Z 332.374,A -85,B 0,C 180,E1 -4422.399,E2 -4422.399} C_VEL
LIN {X 0,Y 532.095,Z 319.98,A -85,B 0,C 180,E1 -4422.927,E2 -4422.927} C_VEL
LIN {X 0,Y 532.296,Z 307.241,A -85,B 0,C 180,E1 -4423.311,E2 -4423.311} C_VEL
LIN {X 0,Y 532.452,Z 293.849,A -85,B 0,C 180,E1 -4423.55,E2 -4423.55} C_VEL
LIN {X 0,Y 532.617,Z 202.426,A -85,B 0,C 180,E1 -4424.793,E2 -4424.793} C_VEL
LIN {X 0,Y 531.217,Z 193.434,A -85,B 0,C 180,E1 -4424.966,E2 -4424.966} C_VEL
LIN {X 0,Y 531.533,Z 176.468,A -85,B 0,C 180,E1 -4427.506,E2 -4427.506} C_VEL
LIN {X 0,Y 531.973,Z 156.558,A -85,B 0,C 180,E1 -4430.519,E2 -4430.519} C_VEL
LIN {X 0,Y 532.251,Z 139.602,A -85,B 0,C 180,E1 -4433.131,E2 -4433.131} C_VEL
LIN {X 0,Y 530.97,Z 132.347,A -85,B 0,C 180,E1 -4434.329,E2 -4434.329} C_VEL
LIN {X 0,Y 530.957,Z 132.345,A -85,B 0,C 180,E1 -4436.746,E2 -4436.746} C_VEL
LIN {X 0,Y 530.964,Z 132.349,A -85,B 0,C 180,E1 -4439.324,E2 -4439.324} C_VEL
LIN {X 0,Y 530.965,Z 132.344,A -85,B 0,C 180,E1 -4442.099,E2 -4442.099} C_VEL
LIN {X 0,Y 530.959,Z 132.342,A -85,B 0,C 180,E1 -4444.849,E2 -4444.849} C_VEL
LIN {X 0,Y 530.964,Z 132.348,A -85,B 0,C 180,E1 -4447.508,E2 -4447.508} C_VEL
LIN {X 0,Y 530.943,Z 132.344,A -85,B 0,C 180,E1 -4450.437,E2 -4450.437} C_VEL
LIN {X 0,Y 530.928,Z 132.349,A -85,B 0,C 180,E1 -4453.499,E2 -4453.499} C_VEL
LIN {X 0,Y 530.967,Z 132.343,A -85,B 0,C 180,E1 -4455.623,E2 -4455.623} C_VEL
LIN {X 0,Y 530.929,Z 132.353,A -85,B 0,C 180,E1 -4458.984,E2 -4458.984} C_VEL
LIN {X 0,Y 530.924,Z 132.347,A -85,B 0,C 180,E1 -4461.526,E2 -4461.526} C_VEL
LIN {X 0,Y 530.925,Z 132.349,A -85,B 0,C 180,E1 -4464.377,E2 -4464.377} C_VEL
LIN {X 0,Y 530.946,Z 132.347,A -85,B 0,C 180,E1 -4467.131,E2 -4467.131} C_VEL
LIN {X 0,Y 530.931,Z 132.344,A -85,B 0,C 180,E1 -4469.8,E2 -4469.8} C_VEL
LIN {X 0,Y 530.956,Z 132.349,A -85,B 0,C 180,E1 -4472.48,E2 -4472.48} C_VEL
LIN {X 0,Y 530.948,Z 132.344,A -85,B 0,C 180,E1 -4475.774,E2 -4475.774} C_VEL
LIN {X 0,Y 530.95,Z 132.347,A -85,B 0,C 180,E1 -4478.245,E2 -4478.245} C_VEL
LIN {X 0,Y 530.919,Z 132.349,A -85,B 0,C 180,E1 -4480.674,E2 -4480.674} C_VEL
LIN {X 0,Y 530.934,Z 132.344,A -85,B 0,C 180,E1 -4483.069,E2 -4483.069} C_VEL
LIN {X 0,Y 531.002,Z 132.337,A -85,B 0,C 180,E1 -4485.435,E2 -4485.435} C_VEL
LIN {X 0,Y 530.99,Z 132.34,A -85,B 0,C 180,E1 -4488.548,E2 -4488.548} C_VEL
LIN {X 0,Y 530.993,Z 132.341,A -85,B 0,C 180,E1 -4491.628,E2 -4491.628} C_VEL
LIN {X 0,Y 531.09,Z 132.325,A -85,B 0,C 180,E1 -4494.685,E2 -4494.685} C_VEL
LIN {X 0,Y 531.138,Z 132.325,A -85,B 0,C 180,E1 -4497.725,E2 -4497.725} C_VEL
LIN {X 0,Y 531.134,Z 132.322,A -85,B 0,C 180,E1 -4500,E2 -4500} C_VEL
LIN {X 0,Y 531.096,Z 132.326,A -85,B 0,C 180,E1 -4503.034,E2 -4503.034} C_VEL
LIN {X 0,Y 531.054,Z 132.329,A -85,B 0,C 180,E1 -4506.077,E2 -4506.077} C_VEL
LIN {X 0,Y 531.015,Z 132.341,A -85,B 0,C 180,E1 -4509.138,E2 -4509.138} C_VEL
LIN {X 0,Y 531.052,Z 132.334,A -85,B 0,C 180,E1 -4511.67,E2 -4511.67} C_VEL
LIN {X 0,Y 531.031,Z 132.337,A -85,B 0,C 180,E1 -4514.954,E2 -4514.954} C_VEL
LIN {X 0,Y 530.982,Z 132.339,A -85,B 0,C 180,E1 -4517.723,E2 -4517.723} C_VEL
LIN {X 0,Y 531.026,Z 132.334,A -85,B 0,C 180,E1 -4520.127,E2 -4520.127} C_VEL
LIN {X 0,Y 530.944,Z 132.346,A -85,B 0,C 180,E1 -4522.573,E2 -4522.573} C_VEL
LIN {X 0,Y 530.97,Z 132.347,A -85,B 0,C 180,E1 -4525.059,E2 -4525.059} C_VEL
LIN {X 0,Y 531.013,Z 132.335,A -85,B 0,C 180,E1 -4527.595,E2 -4527.595} C_VEL
LIN {X 0,Y 530.967,Z 132.349,A -85,B 0,C 180,E1 -4530.643,E2 -4530.643} C_VEL
LIN {X 0,Y 530.962,Z 132.342,A -85,B 0,C 180,E1 -4533.499,E2 -4533.499} C_VEL
LIN {X 0,Y 530.945,Z 132.349,A -85,B 0,C 180,E1 -4536.153,E2 -4536.153} C_VEL
LIN {X 0,Y 530.966,Z 132.347,A -85,B 0,C 180,E1 -4538.653,E2 -4538.653} C_VEL
LIN {X 0,Y 530.996,Z 132.34,A -85,B 0,C 180,E1 -4541.435,E2 -4541.435} C_VEL
LIN {X 0,Y 530.962,Z 132.345,A -85,B 0,C 180,E1 -4543.528,E2 -4543.528} C_VEL
LIN {X 0,Y 530.287,Z 132.434,A -85,B 0,C 180,E1 -4544.162,E2 -4544.162} C_VEL
LIN {X 0,Y 527.439,Z 132.785,A -85,B 0,C 180,E1 -4545.191,E2 -4545.191} C_VEL
LIN {X 0,Y 525.036,Z 133.087,A -85,B 0,C 180,E1 -4546.019,E2 -4546.019} C_VEL
LIN {X 0,Y 524.002,Z 133.213,A -85,B 0,C 180,E1 -4546.658,E2 -4546.658} C_VEL
LIN {X 0,Y 523.917,Z 133.222,A -85,B 0,C 180,E1 -4546.875,E2 -4546.875} C_VEL
LIN {X 0,Y 523.967,Z 133.222,A -85,B 0,C 180,E1 -4549.866,E2 -4549.866} C_VEL
LIN {X 0,Y 523.99,Z 133.289,A -85,B 0,C 180,E1 -4550.3,E2 -4550.3} C_VEL
LIN {X 0,Y 524.526,Z 138.151,A -85,B 0,C 180,E1 -4551.242,E2 -4551.242} C_VEL
LIN {X 0,Y 524.316,Z 153.384,A -85,B 0,C 180,E1 -4554.096,E2 -4554.096} C_VEL
LIN {X 0,Y 524.284,Z 157.946,A -85,B 0,C 180,E1 -4554.91,E2 -4554.91} C_VEL
LIN {X 0,Y 526.038,Z 168.606,A -85,B 0,C 180,E1 -4555.111,E2 -4555.111} C_VEL
LIN {X 0,Y 525.538,Z 264.053,A -85,B 0,C 180,E1 -4556.437,E2 -4556.437} C_VEL
LIN {X 0,Y 525.375,Z 277.023,A -85,B 0,C 180,E1 -4556.765,E2 -4556.765} C_VEL
LIN {X 0,Y 525.145,Z 290.068,A -85,B 0,C 180,E1 -4557.26,E2 -4557.26} C_VEL
LIN {X 0,Y 524.866,Z 301.397,A -85,B 0,C 180,E1 -4557.842,E2 -4557.842} C_VEL
LIN {X 0,Y 524.63,Z 312.56,A -85,B 0,C 180,E1 -4558.584,E2 -4558.584} C_VEL
LIN {X 0,Y 524.332,Z 323.461,A -85,B 0,C 180,E1 -4559.491,E2 -4559.491} C_VEL
LIN {X 0,Y 524.052,Z 333.184,A -85,B 0,C 180,E1 -4560.497,E2 -4560.497} C_VEL
LIN {X 0,Y 523.857,Z 341.461,A -85,B 0,C 180,E1 -4561.558,E2 -4561.558} C_VEL
LIN {X 0,Y 523.697,Z 348.092,A -85,B 0,C 180,E1 -4562.592,E2 -4562.592} C_VEL
LIN {X 0,Y 523.568,Z 353.928,A -85,B 0,C 180,E1 -4563.707,E2 -4563.707} C_VEL
LIN {X 0,Y 523.44,Z 359.185,A -85,B 0,C 180,E1 -4564.98,E2 -4564.98} C_VEL
LIN {X 0,Y 523.361,Z 363.095,A -85,B 0,C 180,E1 -4566.243,E2 -4566.243} C_VEL
LIN {X 0,Y 523.318,Z 365.018,A -85,B 0,C 180,E1 -4567.079,E2 -4567.079} C_VEL
LIN {X 0,Y 523.302,Z 366.443,A -85,B 0,C 180,E1 -4567.921,E2 -4567.921} C_VEL
LIN {X 0,Y 523.284,Z 367.394,A -85,B 0,C 180,E1 -4568.738,E2 -4568.738} C_VEL
LIN {X 0,Y 523.302,Z 367.961,A -85,B 0,C 180,E1 -4570.068,E2 -4570.068} C_VEL
LIN {X 0,Y 523.266,Z 367.511,A -85,B 0,C 180,E1 -4571.195,E2 -4571.195} C_VEL
LIN {X 0,Y 523.307,Z 366.004,A -85,B 0,C 180,E1 -4572.462,E2 -4572.462} C_VEL
LIN {X 0,Y 523.378,Z 362.597,A -85,B 0,C 180,E1 -4574.021,E2 -4574.021} C_VEL
LIN {X 0,Y 523.505,Z 358.75,A -85,B 0,C 180,E1 -4575.222,E2 -4575.222} C_VEL
LIN {X 0,Y 523.571,Z 353.758,A -85,B 0,C 180,E1 -4576.414,E2 -4576.414} C_VEL
LIN {X 0,Y 523.715,Z 347.465,A -85,B 0,C 180,E1 -4577.601,E2 -4577.601} C_VEL
LIN {X 0,Y 523.877,Z 339.58,A -85,B 0,C 180,E1 -4578.788,E2 -4578.788} C_VEL
LIN {X 0,Y 524.13,Z 329.801,A -85,B 0,C 180,E1 -4579.961,E2 -4579.961} C_VEL
LIN {X 0,Y 524.417,Z 319.614,A -85,B 0,C 180,E1 -4580.94,E2 -4580.94} C_VEL
LIN {X 0,Y 524.744,Z 309.204,A -85,B 0,C 180,E1 -4581.741,E2 -4581.741} C_VEL
LIN {X 0,Y 524.995,Z 298.238,A -85,B 0,C 180,E1 -4582.419,E2 -4582.419} C_VEL
LIN {X 0,Y 525.188,Z 286.167,A -85,B 0,C 180,E1 -4582.997,E2 -4582.997} C_VEL
LIN {X 0,Y 525.369,Z 273.749,A -85,B 0,C 180,E1 -4583.423,E2 -4583.423} C_VEL
LIN {X 0,Y 525.534,Z 260.337,A -85,B 0,C 180,E1 -4583.714,E2 -4583.714} C_VEL
LIN {X 0,Y 525.91,Z 166.911,A -85,B 0,C 180,E1 -4585.005,E2 -4585.005} C_VEL
LIN {X 0,Y 524.245,Z 157.614,A -85,B 0,C 180,E1 -4585.194,E2 -4585.194} C_VEL
LIN {X 0,Y 524.478,Z 141.437,A -85,B 0,C 180,E1 -4588.272,E2 -4588.272} C_VEL
LIN {X 0,Y 524.229,Z 134.488,A -85,B 0,C 180,E1 -4589.616,E2 -4589.616} C_VEL
LIN {X 0,Y 524.084,Z 133.207,A -85,B 0,C 180,E1 -4589.904,E2 -4589.904} C_VEL
LIN {X 0,Y 524.099,Z 133.204,A -85,B 0,C 180,E1 -4592.306,E2 -4592.306} C_VEL
LIN {X 0,Y 523.996,Z 133.214,A -85,B 0,C 180,E1 -4596.16,E2 -4596.16} C_VEL
LIN {X 0,Y 523.939,Z 133.217,A -85,B 0,C 180,E1 -4599.263,E2 -4599.263} C_VEL
LIN {X 0,Y 523.923,Z 133.219,A -85,B 0,C 180,E1 -4602.394,E2 -4602.394} C_VEL
LIN {X 0,Y 523.881,Z 133.23,A -85,B 0,C 180,E1 -4605.564,E2 -4605.564} C_VEL
LIN {X 0,Y 523.899,Z 133.225,A -85,B 0,C 180,E1 -4607.972,E2 -4607.972} C_VEL
LIN {X 0,Y 523.899,Z 133.221,A -85,B 0,C 180,E1 -4610.413,E2 -4610.413} C_VEL
LIN {X 0,Y 523.88,Z 133.225,A -85,B 0,C 180,E1 -4612.895,E2 -4612.895} C_VEL
LIN {X 0,Y 523.871,Z 133.233,A -85,B 0,C 180,E1 -4615.423,E2 -4615.423} C_VEL
LIN {X 0,Y 523.892,Z 133.223,A -85,B 0,C 180,E1 -4618.004,E2 -4618.004} C_VEL
LIN {X 0,Y 523.894,Z 133.224,A -85,B 0,C 180,E1 -4620.846,E2 -4620.846} C_VEL
LIN {X 0,Y 523.908,Z 133.222,A -85,B 0,C 180,E1 -4623.727,E2 -4623.727} C_VEL
LIN {X 0,Y 523.855,Z 133.227,A -85,B 0,C 180,E1 -4626.395,E2 -4626.395} C_VEL
LIN {X 0,Y 523.892,Z 133.231,A -85,B 0,C 180,E1 -4629.088,E2 -4629.088} C_VEL
LIN {X 0,Y 523.888,Z 133.222,A -85,B 0,C 180,E1 -4632.126,E2 -4632.126} C_VEL
LIN {X 0,Y 523.932,Z 133.22,A -85,B 0,C 180,E1 -4635.312,E2 -4635.312} C_VEL
LIN {X 0,Y 523.908,Z 133.226,A -85,B 0,C 180,E1 -4638.697,E2 -4638.697} C_VEL
LIN {X 0,Y 523.904,Z 133.225,A -85,B 0,C 180,E1 -4641.083,E2 -4641.083} C_VEL
LIN {X 0,Y 523.862,Z 133.225,A -85,B 0,C 180,E1 -4643.823,E2 -4643.823} C_VEL
LIN {X 0,Y 523.896,Z 133.23,A -85,B 0,C 180,E1 -4646.633,E2 -4646.633} C_VEL
LIN {X 0,Y 523.907,Z 133.22,A -85,B 0,C 180,E1 -4649.353,E2 -4649.353} C_VEL
LIN {X 0,Y 523.912,Z 133.225,A -85,B 0,C 180,E1 -4652.296,E2 -4652.296} C_VEL
LIN {X 0,Y 523.899,Z 133.221,A -85,B 0,C 180,E1 -4655.427,E2 -4655.427} C_VEL
LIN {X 0,Y 523.922,Z 133.221,A -85,B 0,C 180,E1 -4657.939,E2 -4657.939} C_VEL
LIN {X 0,Y 523.902,Z 133.228,A -85,B 0,C 180,E1 -4660.406,E2 -4660.406} C_VEL
LIN {X 0,Y 523.902,Z 133.222,A -85,B 0,C 180,E1 -4662.836,E2 -4662.836} C_VEL
LIN {X 0,Y 523.905,Z 133.227,A -85,B 0,C 180,E1 -4666.028,E2 -4666.028} C_VEL
LIN {X 0,Y 523.964,Z 133.218,A -85,B 0,C 180,E1 -4668.393,E2 -4668.393} C_VEL
LIN {X 0,Y 523.949,Z 133.217,A -85,B 0,C 180,E1 -4671.516,E2 -4671.516} C_VEL
LIN {X 0,Y 524.031,Z 133.205,A -85,B 0,C 180,E1 -4674.614,E2 -4674.614} C_VEL
LIN {X 0,Y 524.107,Z 133.201,A -85,B 0,C 180,E1 -4677.695,E2 -4677.695} C_VEL
LIN {X 0,Y 524.1,Z 133.202,A -85,B 0,C 180,E1 -4680,E2 -4680} C_VEL
LIN {X 0,Y 524.106,Z 133.197,A -85,B 0,C 180,E1 -4682.306,E2 -4682.306} C_VEL
LIN {X 0,Y 524.001,Z 133.211,A -85,B 0,C 180,E1 -4686.16,E2 -4686.16} C_VEL
LIN {X 0,Y 523.951,Z 133.218,A -85,B 0,C 180,E1 -4689.263,E2 -4689.263} C_VEL
LIN {X 0,Y 524.003,Z 133.214,A -85,B 0,C 180,E1 -4691.736,E2 -4691.736} C_VEL
LIN {X 0,Y 523.988,Z 133.213,A -85,B 0,C 180,E1 -4695.048,E2 -4695.048} C_VEL
LIN {X 0,Y 523.919,Z 133.22,A -85,B 0,C 180,E1 -4697.971,E2 -4697.971} C_VEL
LIN {X 0,Y 523.944,Z 133.215,A -85,B 0,C 180,E1 -4700.412,E2 -4700.412} C_VEL
LIN {X 0,Y 523.892,Z 133.225,A -85,B 0,C 180,E1 -4702.895,E2 -4702.895} C_VEL
LIN {X 0,Y 523.902,Z 133.226,A -85,B 0,C 180,E1 -4705.422,E2 -4705.422} C_VEL
LIN {X 0,Y 523.901,Z 133.221,A -85,B 0,C 180,E1 -4708.003,E2 -4708.003} C_VEL
LIN {X 0,Y 523.903,Z 133.226,A -85,B 0,C 180,E1 -4710.846,E2 -4710.846} C_VEL
LIN {X 0,Y 523.931,Z 133.217,A -85,B 0,C 180,E1 -4713.729,E2 -4713.729} C_VEL
LIN {X 0,Y 523.902,Z 133.222,A -85,B 0,C 180,E1 -4716.4,E2 -4716.4} C_VEL
LIN {X 0,Y 523.916,Z 133.224,A -85,B 0,C 180,E1 -4719.086,E2 -4719.086} C_VEL
LIN {X 0,Y 523.903,Z 133.221,A -85,B 0,C 180,E1 -4722.124,E2 -4722.124} C_VEL
LIN {X 0,Y 523.938,Z 133.217,A -85,B 0,C 180,E1 -4725.311,E2 -4725.311} C_VEL
LIN {X 0,Y 523.924,Z 133.226,A -85,B 0,C 180,E1 -4728.694,E2 -4728.694} C_VEL
LIN {X 0,Y 523.914,Z 133.22,A -85,B 0,C 180,E1 -4731.898,E2 -4731.898} C_VEL
LIN {X 0,Y 523.921,Z 133.221,A -85,B 0,C 180,E1 -4734.912,E2 -4734.912} C_VEL
LIN {X 0,Y 523.938,Z 133.217,A -85,B 0,C 180,E1 -4737.68,E2 -4737.68} C_VEL
LIN {X 0,Y 523.939,Z 133.221,A -85,B 0,C 180,E1 -4740.68,E2 -4740.68} C_VEL
LIN {X 0,Y 523.906,Z 133.226,A -85,B 0,C 180,E1 -4743.724,E2 -4743.724} C_VEL
LIN {X 0,Y 523.947,Z 133.345,A -85,B 0,C 180,E1 -4745.48,E2 -4745.48} C_VEL
LIN {X 0,Y 525.316,Z 140.963,A -85,B 0,C 180,E1 -4746.754,E2 -4746.754} C_VEL
LIN {X 0,Y 525.058,Z 156.738,A -85,B 0,C 180,E1 -4749.225,E2 -4749.225} C_VEL
LIN {X 0,Y 524.559,Z 177.701,A -85,B 0,C 180,E1 -4752.455,E2 -4752.455} C_VEL
LIN {X 0,Y 524.253,Z 193.503,A -85,B 0,C 180,E1 -4754.844,E2 -4754.844} C_VEL
LIN {X 0,Y 525.876,Z 204.971,A -85,B 0,C 180,E1 -4755.051,E2 -4755.051} C_VEL
LIN {X 0,Y 525.476,Z 302.516,A -85,B 0,C 180,E1 -4756.415,E2 -4756.415} C_VEL
LIN {X 0,Y 525.232,Z 316.287,A -85,B 0,C 180,E1 -4756.778,E2 -4756.778} C_VEL
LIN {X 0,Y 524.974,Z 329.159,A -85,B 0,C 180,E1 -4757.288,E2 -4757.288} C_VEL
LIN {X 0,Y 524.666,Z 341.762,A -85,B 0,C 180,E1 -4757.971,E2 -4757.971} C_VEL
LIN {X 0,Y 524.461,Z 352.265,A -85,B 0,C 180,E1 -4758.698,E2 -4758.698} C_VEL
LIN {X 0,Y 524.158,Z 362.494,A -85,B 0,C 180,E1 -4759.571,E2 -4759.571} C_VEL
LIN {X 0,Y 523.935,Z 371.695,A -85,B 0,C 180,E1 -4760.542,E2 -4760.542} C_VEL
LIN {X 0,Y 523.717,Z 380.659,A -85,B 0,C 180,E1 -4761.705,E2 -4761.705} C_VEL
LIN {X 0,Y 523.569,Z 387.875,A -85,B 0,C 180,E1 -4762.867,E2 -4762.867} C_VEL
LIN {X 0,Y 523.461,Z 392.744,A -85,B 0,C 180,E1 -4763.834,E2 -4763.834} C_VEL
LIN {X 0,Y 523.383,Z 397.476,A -85,B 0,C 180,E1 -4764.993,E2 -4764.993} C_VEL
LIN {X 0,Y 523.443,Z 401.096,A -85,B 0,C 180,E1 -4766.151,E2 -4766.151} C_VEL
LIN {X 0,Y 523.368,Z 402.958,A -85,B 0,C 180,E1 -4766.921,E2 -4766.921} C_VEL
LIN {X 0,Y 523.335,Z 404.356,A -85,B 0,C 180,E1 -4767.691,E2 -4767.691} C_VEL
LIN {X 0,Y 523.256,Z 405.959,A -85,B 0,C 180,E1 -4769.23,E2 -4769.23} C_VEL
LIN {X 0,Y 523.257,Z 406.174,A -85,B 0,C 180,E1 -4770,E2 -4770} C_VEL
LIN {X 0,Y 523.275,Z 405.348,A -85,B 0,C 180,E1 -4771.539,E2 -4771.539} C_VEL
LIN {X 0,Y 523.335,Z 404.351,A -85,B 0,C 180,E1 -4772.309,E2 -4772.309} C_VEL
LIN {X 0,Y 523.368,Z 402.951,A -85,B 0,C 180,E1 -4773.079,E2 -4773.079} C_VEL
LIN {X 0,Y 523.422,Z 400.008,A -85,B 0,C 180,E1 -4774.235,E2 -4774.235} C_VEL
LIN {X 0,Y 523.456,Z 396.022,A -85,B 0,C 180,E1 -4775.393,E2 -4775.393} C_VEL
LIN {X 0,Y 523.503,Z 389.967,A -85,B 0,C 180,E1 -4776.731,E2 -4776.731} C_VEL
LIN {X 0,Y 523.644,Z 383.195,A -85,B 0,C 180,E1 -4777.907,E2 -4777.907} C_VEL
LIN {X 0,Y 523.827,Z 374.885,A -85,B 0,C 180,E1 -4779.07,E2 -4779.07} C_VEL
LIN {X 0,Y 524.028,Z 366.366,A -85,B 0,C 180,E1 -4780.041,E2 -4780.041} C_VEL
LIN {X 0,Y 524.316,Z 355.843,A -85,B 0,C 180,E1 -4781.012,E2 -4781.012} C_VEL
LIN {X 0,Y 524.595,Z 345.618,A -85,B 0,C 180,E1 -4781.776,E2 -4781.776} C_VEL
LIN {X 0,Y 524.887,Z 334.018,A -85,B 0,C 180,E1 -4782.469,E2 -4782.469} C_VEL
